LIN {X -91.168,Y -9.449,Z -75.108,A -90.000,B 90.000,C 0.000} C_DIS
LIN {X -91.268,Y -9.455,Z -75.087,A -90.000,B 90.000,C 0.000} C_DIS
LIN {X -91.699,Y -9.484,Z -75.022,A -90.000,B 90.000,C 0.000} C_DIS
LIN {X -91.909,Y -9.497,Z -74.992,A -90.000,B 90.000,C 0.000} C_DIS
LIN {X -92.204,Y -9.516,Z -74.968,A -90.000,B 90.000,C 0.000} C_DIS
LIN {X -92.548,Y -9.529,Z -74.936,A -90.000,B 90.000,C 0.000} C_DIS
LIN {X -93.104,Y -9.554,Z -74.909,A -90.000,B 90.000,C 0.000} C_DIS
LIN {X -93.295,Y -9.561,Z -74.896,A -90.000,B 90.000,C 0.000} C_DIS
LIN {X -93.565,Y -9.563,Z -74.882,A -90.000,B 90.000,C 0.000} C_DIS
LIN {X -93.812,Y -9.568,Z -74.866,A -90.000,B 90.000,C 0.000} C_DIS
LIN {X -94.175,Y -9.581,Z -74.843,A -90.000,B 90.000,C 0.000} C_DIS
LIN {X -94.333,Y -9.590,Z -74.840,A -90.000,B 90.000,C 0.000} C_DIS
LIN {X -94.789,Y -9.599,Z -74.813,A -90.000,B 90.000,C 0.000} C_DIS
LIN {X -95.233,Y -9.601,Z -74.772,A -90.000,B 90.000,C 0.000} C_DIS
LIN {X -95.684,Y -9.621,Z -74.743,A -90.000,B 90.000,C 0.000} C_DIS
LIN {X -95.934,Y -9.627,Z -74.715,A -90.000,B 90.000,C 0.000} C_DIS
LIN {X -95.995,Y -9.627,Z -74.706,A -90.000,B 90.000,C 0.000} C_DIS
LIN {X -96.123,Y -9.624,Z -74.688,A -90.000,B 90.000,C 0.000} C_DIS
LIN {X -96.497,Y -9.616,Z -74.630,A -90.000,B 90.000,C 0.000} C_DIS
LIN {X -96.581,Y -9.616,Z -74.619,A -90.000,B 90.000,C 0.000} C_DIS
LIN {X -96.934,Y -9.624,Z -74.567,A -90.000,B 90.000,C 0.000} C_DIS
LIN {X -97.349,Y -9.643,Z -74.499,A -90.000,B 90.000,C 0.000} C_DIS
LIN {X -97.387,Y -9.643,Z -74.491,A -90.000,B 90.000,C 0.000} C_DIS
LIN {X -97.586,Y -9.638,Z -74.449,A -90.000,B 90.000,C 0.000} C_DIS
LIN {X -97.776,Y -9.630,Z -74.406,A -90.000,B 90.000,C 0.000} C_DIS
LIN {X -97.980,Y -9.623,Z -74.352,A -90.000,B 90.000,C 0.000} C_DIS
LIN {X -98.394,Y -9.618,Z -74.242,A -90.000,B 90.000,C 0.000} C_DIS
LIN {X -98.720,Y -9.626,Z -74.148,A -90.000,B 90.000,C 0.000} C_DIS
LIN {X -99.033,Y -9.638,Z -74.054,A -90.000,B 90.000,C 0.000} C_DIS
LIN {X -99.091,Y -9.639,Z -74.038,A -90.000,B 90.000,C 0.000} C_DIS
LIN {X -99.335,Y -9.635,Z -73.957,A -90.000,B 90.000,C 0.000} C_DIS
LIN {X -99.558,Y -9.626,Z -73.875,A -90.000,B 90.000,C 0.000} C_DIS
LIN {X -99.757,Y -9.620,Z -73.799,A -90.000,B 90.000,C 0.000} C_DIS
LIN {X -100.008,Y -9.607,Z -73.687,A -90.000,B 90.000,C 0.000} C_DIS
LIN {X -100.150,Y -9.603,Z -73.626,A -90.000,B 90.000,C 0.000} C_DIS
LIN {X -100.449,Y -9.604,Z -73.493,A -90.000,B 90.000,C 0.000} C_DIS
LIN {X -100.910,Y -9.619,Z -73.278,A -90.000,B 90.000,C 0.000} C_DIS
LIN {X -101.101,Y -9.624,Z -73.186,A -90.000,B 90.000,C 0.000} C_DIS
LIN {X -101.527,Y -9.617,Z -72.967,A -90.000,B 90.000,C 0.000} C_DIS
LIN {X -101.902,Y -9.589,Z -72.732,A -90.000,B 90.000,C 0.000} C_DIS
LIN {X -101.991,Y -9.585,Z -72.673,A -90.000,B 90.000,C 0.000} C_DIS
LIN {X -102.294,Y -9.577,Z -72.481,A -90.000,B 90.000,C 0.000} C_DIS
LIN {X -102.915,Y -9.585,Z -72.073,A -90.000,B 90.000,C 0.000} C_DIS
LIN {X -103.087,Y -9.586,Z -71.956,A -90.000,B 90.000,C 0.000} C_DIS
LIN {X -103.329,Y -9.590,Z -71.789,A -90.000,B 90.000,C 0.000} C_DIS
LIN {X -104.055,Y -9.563,Z -71.187,A -90.000,B 90.000,C 0.000} C_DIS
LIN {X -104.727,Y -9.571,Z -70.630,A -90.000,B 90.000,C 0.000} C_DIS
LIN {X -105.073,Y -9.578,Z -70.329,A -90.000,B 90.000,C 0.000} C_DIS
LIN {X -105.804,Y -9.557,Z -69.596,A -90.000,B 90.000,C 0.000} C_DIS
LIN {X -106.031,Y -9.558,Z -69.362,A -90.000,B 90.000,C 0.000} C_DIS
LIN {X -106.363,Y -9.567,Z -69.030,A -90.000,B 90.000,C 0.000} C_DIS
LIN {X -106.675,Y -9.569,Z -68.696,A -90.000,B 90.000,C 0.000} C_DIS
LIN {X -107.151,Y -9.555,Z -68.140,A -90.000,B 90.000,C 0.000} C_DIS
LIN {X -107.437,Y -9.551,Z -67.804,A -90.000,B 90.000,C 0.000} C_DIS
LIN {X -107.704,Y -9.554,Z -67.487,A -90.000,B 90.000,C 0.000} C_DIS
LIN {X -107.793,Y -9.554,Z -67.378,A -90.000,B 90.000,C 0.000} C_DIS
LIN {X -108.035,Y -9.548,Z -67.063,A -90.000,B 90.000,C 0.000} C_DIS
LIN {X -108.277,Y -9.542,Z -66.740,A -90.000,B 90.000,C 0.000} C_DIS
LIN {X -108.656,Y -9.536,Z -66.235,A -90.000,B 90.000,C 0.000} C_DIS
LIN {X -109.055,Y -9.536,Z -65.697,A -90.000,B 90.000,C 0.000} C_DIS
LIN {X -109.521,Y -9.515,Z -64.985,A -90.000,B 90.000,C 0.000} C_DIS
LIN {X -109.784,Y -9.507,Z -64.583,A -90.000,B 90.000,C 0.000} C_DIS
LIN {X -109.990,Y -9.509,Z -64.262,A -90.000,B 90.000,C 0.000} C_DIS
LIN {X -110.250,Y -9.507,Z -63.841,A -90.000,B 90.000,C 0.000} C_DIS
LIN {X -110.475,Y -9.498,Z -63.445,A -90.000,B 90.000,C 0.000} C_DIS
LIN {X -110.954,Y -9.484,Z -62.593,A -90.000,B 90.000,C 0.000} C_DIS
LIN {X -111.235,Y -9.477,Z -62.028,A -90.000,B 90.000,C 0.000} C_DIS
LIN {X -111.470,Y -9.467,Z -61.530,A -90.000,B 90.000,C 0.000} C_DIS
LIN {X -111.674,Y -9.468,Z -61.087,A -90.000,B 90.000,C 0.000} C_DIS
LIN {X -111.779,Y -9.472,Z -60.856,A -90.000,B 90.000,C 0.000} C_DIS
LIN {X -111.969,Y -9.471,Z -60.371,A -90.000,B 90.000,C 0.000} C_DIS
LIN {X -112.195,Y -9.468,Z -59.781,A -90.000,B 90.000,C 0.000} C_DIS
LIN {X -112.476,Y -9.471,Z -59.008,A -90.000,B 90.000,C 0.000} C_DIS
LIN {X -112.532,Y -9.474,Z -58.843,A -90.000,B 90.000,C 0.000} C_DIS
LIN {X -112.797,Y -9.477,Z -57.968,A -90.000,B 90.000,C 0.000} C_DIS
LIN {X -112.866,Y -9.485,Z -57.732,A -90.000,B 90.000,C 0.000} C_DIS
LIN {X -112.980,Y -9.499,Z -57.320,A -90.000,B 90.000,C 0.000} C_DIS
LIN {X -113.114,Y -9.515,Z -56.783,A -90.000,B 90.000,C 0.000} C_DIS
LIN {X -113.186,Y -9.521,Z -56.488,A -90.000,B 90.000,C 0.000} C_DIS
LIN {X -113.300,Y -9.536,Z -56.059,A -90.000,B 90.000,C 0.000} C_DIS
LIN {X -113.345,Y -9.541,Z -55.892,A -90.000,B 90.000,C 0.000} C_DIS
LIN {X -113.481,Y -9.549,Z -55.371,A -90.000,B 90.000,C 0.000} C_DIS
LIN {X -113.611,Y -9.568,Z -54.950,A -90.000,B 90.000,C 0.000} C_DIS
LIN {X -113.730,Y -9.575,Z -54.580,A -90.000,B 90.000,C 0.000} C_DIS
LIN {X -113.845,Y -9.584,Z -54.240,A -90.000,B 90.000,C 0.000} C_DIS
LIN {X -113.948,Y -9.588,Z -53.949,A -90.000,B 90.000,C 0.000} C_DIS
LIN {X -114.127,Y -9.591,Z -53.418,A -90.000,B 90.000,C 0.000} C_DIS
LIN {X -114.176,Y -9.591,Z -53.268,A -90.000,B 90.000,C 0.000} C_DIS
LIN {X -114.354,Y -9.592,Z -52.715,A -90.000,B 90.000,C 0.000} C_DIS
LIN {X -114.494,Y -9.589,Z -52.161,A -90.000,B 90.000,C 0.000} C_DIS
LIN {X -114.530,Y -9.591,Z -52.010,A -90.000,B 90.000,C 0.000} C_DIS
LIN {X -114.581,Y -9.592,Z -51.768,A -90.000,B 90.000,C 0.000} C_DIS
LIN {X -114.638,Y -9.569,Z -51.559,A -90.000,B 90.000,C 0.000} C_DIS
LIN {X -114.665,Y -9.552,Z -51.423,A -90.000,B 90.000,C 0.000} C_DIS
LIN {X -114.732,Y -9.507,Z -51.064,A -90.000,B 90.000,C 0.000} C_DIS
LIN {X -114.755,Y -9.494,Z -50.930,A -90.000,B 90.000,C 0.000} C_DIS
LIN {X -114.825,Y -9.450,Z -50.470,A -90.000,B 90.000,C 0.000} C_DIS
LIN {X -114.863,Y -9.414,Z -50.095,A -90.000,B 90.000,C 0.000} C_DIS
LIN {X -114.873,Y -9.404,Z -49.977,A -90.000,B 90.000,C 0.000} C_DIS
LIN {X -115.001,Y -9.414,Z -49.692,A -90.000,B 90.000,C 0.000} C_DIS
LIN {X -115.085,Y -9.419,Z -49.499,A -90.000,B 90.000,C 0.000} C_DIS
LIN {X -115.200,Y -9.434,Z -49.219,A -90.000,B 90.000,C 0.000} C_DIS
LIN {X -115.364,Y -9.456,Z -48.784,A -90.000,B 90.000,C 0.000} C_DIS
LIN {X -115.419,Y -9.463,Z -48.623,A -90.000,B 90.000,C 0.000} C_DIS
LIN {X -115.494,Y -9.476,Z -48.397,A -90.000,B 90.000,C 0.000} C_DIS
LIN {X -115.570,Y -9.486,Z -48.140,A -90.000,B 90.000,C 0.000} C_DIS
LIN {X -115.656,Y -9.511,Z -47.832,A -90.000,B 90.000,C 0.000} C_DIS
LIN {X -115.783,Y -9.545,Z -47.228,A -90.000,B 90.000,C 0.000} C_DIS
LIN {X -115.820,Y -9.560,Z -47.041,A -90.000,B 90.000,C 0.000} C_DIS
LIN {X -115.835,Y -9.566,Z -46.935,A -90.000,B 90.000,C 0.000} C_DIS
LIN {X -115.860,Y -9.577,Z -46.716,A -90.000,B 90.000,C 0.000} C_DIS
LIN {X -115.875,Y -9.588,Z -46.570,A -90.000,B 90.000,C 0.000} C_DIS
LIN {X -115.897,Y -9.607,Z -46.245,A -90.000,B 90.000,C 0.000} C_DIS
LIN {X -115.918,Y -9.644,Z -45.793,A -90.000,B 90.000,C 0.000} C_DIS
LIN {X -115.894,Y -9.672,Z -45.327,A -90.000,B 90.000,C 0.000} C_DIS
LIN {X -115.872,Y -9.694,Z -45.037,A -90.000,B 90.000,C 0.000} C_DIS
LIN {X -115.826,Y -9.720,Z -44.669,A -90.000,B 90.000,C 0.000} C_DIS
LIN {X -115.752,Y -9.743,Z -44.251,A -90.000,B 90.000,C 0.000} C_DIS
LIN {X -115.713,Y -9.747,Z -44.091,A -90.000,B 90.000,C 0.000} C_DIS
LIN {X -115.664,Y -9.757,Z -43.912,A -90.000,B 90.000,C 0.000} C_DIS
LIN {X -115.614,Y -9.765,Z -43.739,A -90.000,B 90.000,C 0.000} C_DIS
LIN {X -115.524,Y -9.782,Z -43.444,A -90.000,B 90.000,C 0.000} C_DIS
LIN {X -115.525,Y -9.755,Z -43.363,A -90.000,B 90.000,C 0.000} C_DIS
LIN {X -115.523,Y -9.708,Z -43.212,A -90.000,B 90.000,C 0.000} C_DIS
LIN {X -115.512,Y -9.657,Z -43.054,A -90.000,B 90.000,C 0.000} C_DIS
LIN {X -115.504,Y -9.620,Z -42.928,A -90.000,B 90.000,C 0.000} C_DIS
LIN {X -115.490,Y -9.576,Z -42.771,A -90.000,B 90.000,C 0.000} C_DIS
LIN {X -115.474,Y -9.541,Z -42.647,A -90.000,B 90.000,C 0.000} C_DIS
LIN {X -115.434,Y -9.476,Z -42.387,A -90.000,B 90.000,C 0.000} C_DIS
LIN {X -115.413,Y -9.451,Z -42.272,A -90.000,B 90.000,C 0.000} C_DIS
LIN {X -115.362,Y -9.404,Z -42.049,A -90.000,B 90.000,C 0.000} C_DIS
LIN {X -115.335,Y -9.385,Z -41.942,A -90.000,B 90.000,C 0.000} C_DIS
LIN {X -115.562,Y -9.395,Z -41.403,A -90.000,B 90.000,C 0.000} C_DIS
LIN {X -115.834,Y -9.409,Z -40.701,A -90.000,B 90.000,C 0.000} C_DIS
LIN {X -115.898,Y -9.411,Z -40.527,A -90.000,B 90.000,C 0.000} C_DIS
LIN {X -115.998,Y -9.421,Z -40.242,A -90.000,B 90.000,C 0.000} C_DIS
LIN {X -116.124,Y -9.434,Z -39.859,A -90.000,B 90.000,C 0.000} C_DIS
LIN {X -116.188,Y -9.437,Z -39.625,A -90.000,B 90.000,C 0.000} C_DIS
LIN {X -116.280,Y -9.448,Z -39.279,A -90.000,B 90.000,C 0.000} C_DIS
LIN {X -116.338,Y -9.459,Z -39.055,A -90.000,B 90.000,C 0.000} C_DIS
LIN {X -116.435,Y -9.475,Z -38.570,A -90.000,B 90.000,C 0.000} C_DIS
LIN {X -116.495,Y -9.485,Z -38.207,A -90.000,B 90.000,C 0.000} C_DIS
LIN {X -116.519,Y -9.488,Z -38.006,A -90.000,B 90.000,C 0.000} C_DIS
LIN {X -116.557,Y -9.499,Z -37.661,A -90.000,B 90.000,C 0.000} C_DIS
LIN {X -116.577,Y -9.508,Z -37.467,A -90.000,B 90.000,C 0.000} C_DIS
LIN {X -116.590,Y -9.517,Z -37.185,A -90.000,B 90.000,C 0.000} C_DIS
LIN {X -116.592,Y -9.520,Z -37.070,A -90.000,B 90.000,C 0.000} C_DIS
LIN {X -116.593,Y -9.528,Z -36.748,A -90.000,B 90.000,C 0.000} C_DIS
LIN {X -116.588,Y -9.536,Z -36.577,A -90.000,B 90.000,C 0.000} C_DIS
LIN {X -116.583,Y -9.544,Z -36.410,A -90.000,B 90.000,C 0.000} C_DIS
LIN {X -116.566,Y -9.555,Z -36.116,A -90.000,B 90.000,C 0.000} C_DIS
LIN {X -116.555,Y -9.557,Z -35.992,A -90.000,B 90.000,C 0.000} C_DIS
LIN {X -116.518,Y -9.569,Z -35.688,A -90.000,B 90.000,C 0.000} C_DIS
LIN {X -116.455,Y -9.588,Z -35.269,A -90.000,B 90.000,C 0.000} C_DIS
LIN {X -116.407,Y -9.596,Z -35.023,A -90.000,B 90.000,C 0.000} C_DIS
LIN {X -116.292,Y -9.604,Z -34.552,A -90.000,B 90.000,C 0.000} C_DIS
LIN {X -116.219,Y -9.613,Z -34.281,A -90.000,B 90.000,C 0.000} C_DIS
LIN {X -116.131,Y -9.620,Z -34.013,A -90.000,B 90.000,C 0.000} C_DIS
LIN {X -115.955,Y -9.626,Z -33.530,A -90.000,B 90.000,C 0.000} C_DIS
LIN {X -115.874,Y -9.632,Z -33.322,A -90.000,B 90.000,C 0.000} C_DIS
LIN {X -115.828,Y -9.634,Z -33.217,A -90.000,B 90.000,C 0.000} C_DIS
LIN {X -115.781,Y -9.638,Z -33.111,A -90.000,B 90.000,C 0.000} C_DIS
LIN {X -115.641,Y -9.647,Z -32.806,A -90.000,B 90.000,C 0.000} C_DIS
LIN {X -115.507,Y -9.653,Z -32.547,A -90.000,B 90.000,C 0.000} C_DIS
LIN {X -115.409,Y -9.659,Z -32.366,A -90.000,B 90.000,C 0.000} C_DIS
LIN {X -115.298,Y -9.671,Z -32.168,A -90.000,B 90.000,C 0.000} C_DIS
LIN {X -115.155,Y -9.677,Z -31.942,A -90.000,B 90.000,C 0.000} C_DIS
LIN {X -114.995,Y -9.683,Z -31.708,A -90.000,B 90.000,C 0.000} C_DIS
LIN {X -114.890,Y -9.691,Z -31.560,A -90.000,B 90.000,C 0.000} C_DIS
LIN {X -114.702,Y -9.699,Z -31.322,A -90.000,B 90.000,C 0.000} C_DIS
LIN {X -114.414,Y -9.707,Z -30.991,A -90.000,B 90.000,C 0.000} C_DIS
LIN {X -114.202,Y -9.712,Z -30.773,A -90.000,B 90.000,C 0.000} C_DIS
LIN {X -113.932,Y -9.710,Z -30.509,A -90.000,B 90.000,C 0.000} C_DIS
LIN {X -113.798,Y -9.696,Z -30.361,A -90.000,B 90.000,C 0.000} C_DIS
LIN {X -113.705,Y -9.684,Z -30.257,A -90.000,B 90.000,C 0.000} C_DIS
LIN {X -113.657,Y -9.679,Z -30.199,A -90.000,B 90.000,C 0.000} C_DIS
LIN {X -113.484,Y -9.675,Z -29.956,A -90.000,B 90.000,C 0.000} C_DIS
LIN {X -113.219,Y -9.679,Z -29.558,A -90.000,B 90.000,C 0.000} C_DIS
LIN {X -112.886,Y -9.691,Z -29.072,A -90.000,B 90.000,C 0.000} C_DIS
LIN {X -112.575,Y -9.712,Z -28.647,A -90.000,B 90.000,C 0.000} C_DIS
LIN {X -112.441,Y -9.714,Z -28.475,A -90.000,B 90.000,C 0.000} C_DIS
LIN {X -112.214,Y -9.724,Z -28.195,A -90.000,B 90.000,C 0.000} C_DIS
LIN {X -111.965,Y -9.730,Z -27.908,A -90.000,B 90.000,C 0.000} C_DIS
LIN {X -111.767,Y -9.733,Z -27.682,A -90.000,B 90.000,C 0.000} C_DIS
LIN {X -111.552,Y -9.744,Z -27.448,A -90.000,B 90.000,C 0.000} C_DIS
LIN {X -111.335,Y -9.745,Z -27.227,A -90.000,B 90.000,C 0.000} C_DIS
LIN {X -111.169,Y -9.752,Z -27.063,A -90.000,B 90.000,C 0.000} C_DIS
LIN {X -110.868,Y -9.756,Z -26.783,A -90.000,B 90.000,C 0.000} C_DIS
LIN {X -110.555,Y -9.759,Z -26.498,A -90.000,B 90.000,C 0.000} C_DIS
LIN {X -110.409,Y -9.764,Z -26.368,A -90.000,B 90.000,C 0.000} C_DIS
LIN {X -110.072,Y -9.763,Z -26.089,A -90.000,B 90.000,C 0.000} C_DIS
LIN {X -109.993,Y -9.765,Z -26.026,A -90.000,B 90.000,C 0.000} C_DIS
LIN {X -109.797,Y -9.772,Z -25.877,A -90.000,B 90.000,C 0.000} C_DIS
LIN {X -109.647,Y -9.773,Z -25.770,A -90.000,B 90.000,C 0.000} C_DIS
LIN {X -109.156,Y -9.772,Z -25.430,A -90.000,B 90.000,C 0.000} C_DIS
LIN {X -109.060,Y -9.773,Z -25.365,A -90.000,B 90.000,C 0.000} C_DIS
LIN {X -108.938,Y -9.779,Z -25.289,A -90.000,B 90.000,C 0.000} C_DIS
LIN {X -108.645,Y -9.778,Z -25.128,A -90.000,B 90.000,C 0.000} C_DIS
LIN {X -107.965,Y -9.778,Z -24.760,A -90.000,B 90.000,C 0.000} C_DIS
LIN {X -107.894,Y -9.777,Z -24.729,A -90.000,B 90.000,C 0.000} C_DIS
LIN {X -107.430,Y -9.777,Z -24.533,A -90.000,B 90.000,C 0.000} C_DIS
LIN {X -107.064,Y -9.775,Z -24.380,A -90.000,B 90.000,C 0.000} C_DIS
LIN {X -106.859,Y -9.774,Z -24.300,A -90.000,B 90.000,C 0.000} C_DIS
LIN {X -106.675,Y -9.768,Z -24.235,A -90.000,B 90.000,C 0.000} C_DIS
LIN {X -105.951,Y -9.767,Z -23.999,A -90.000,B 90.000,C 0.000} C_DIS
LIN {X -105.833,Y -9.766,Z -23.963,A -90.000,B 90.000,C 0.000} C_DIS
LIN {X -105.591,Y -9.759,Z -23.893,A -90.000,B 90.000,C 0.000} C_DIS
LIN {X -104.540,Y -9.751,Z -23.612,A -90.000,B 90.000,C 0.000} C_DIS
LIN {X -104.007,Y -9.738,Z -23.487,A -90.000,B 90.000,C 0.000} C_DIS
LIN {X -103.457,Y -9.732,Z -23.351,A -90.000,B 90.000,C 0.000} C_DIS
LIN {X -102.983,Y -9.716,Z -23.250,A -90.000,B 90.000,C 0.000} C_DIS
LIN {X -102.872,Y -9.662,Z -23.190,A -90.000,B 90.000,C 0.000} C_DIS
LIN {X -102.791,Y -9.626,Z -23.147,A -90.000,B 90.000,C 0.000} C_DIS
LIN {X -102.651,Y -9.570,Z -23.076,A -90.000,B 90.000,C 0.000} C_DIS
LIN {X -102.484,Y -9.509,Z -22.997,A -90.000,B 90.000,C 0.000} C_DIS
LIN {X -102.347,Y -9.465,Z -22.940,A -90.000,B 90.000,C 0.000} C_DIS
LIN {X -102.173,Y -9.419,Z -22.874,A -90.000,B 90.000,C 0.000} C_DIS
LIN {X -102.051,Y -9.391,Z -22.833,A -90.000,B 90.000,C 0.000} C_DIS
LIN {X -101.981,Y -9.396,Z -22.678,A -90.000,B 90.000,C 0.000} C_DIS
LIN {X -101.915,Y -9.397,Z -22.554,A -90.000,B 90.000,C 0.000} C_DIS
LIN {X -101.706,Y -9.412,Z -22.179,A -90.000,B 90.000,C 0.000} C_DIS
LIN {X -101.652,Y -9.413,Z -22.097,A -90.000,B 90.000,C 0.000} C_DIS
LIN {X -101.407,Y -9.417,Z -21.742,A -90.000,B 90.000,C 0.000} C_DIS
LIN {X -101.220,Y -9.429,Z -21.478,A -90.000,B 90.000,C 0.000} C_DIS
LIN {X -101.124,Y -9.431,Z -21.364,A -90.000,B 90.000,C 0.000} C_DIS
LIN {X -100.916,Y -9.439,Z -21.124,A -90.000,B 90.000,C 0.000} C_DIS
LIN {X -100.729,Y -9.441,Z -20.929,A -90.000,B 90.000,C 0.000} C_DIS
LIN {X -100.489,Y -9.453,Z -20.691,A -90.000,B 90.000,C 0.000} C_DIS
LIN {X -100.427,Y -9.456,Z -20.633,A -90.000,B 90.000,C 0.000} C_DIS
LIN {X -100.372,Y -9.456,Z -20.587,A -90.000,B 90.000,C 0.000} C_DIS
LIN {X -100.028,Y -9.469,Z -20.310,A -90.000,B 90.000,C 0.000} C_DIS
LIN {X -99.660,Y -9.482,Z -20.039,A -90.000,B 90.000,C 0.000} C_DIS
LIN {X -99.572,Y -9.484,Z -19.982,A -90.000,B 90.000,C 0.000} C_DIS
LIN {X -99.263,Y -9.501,Z -19.787,A -90.000,B 90.000,C 0.000} C_DIS
LIN {X -99.057,Y -9.514,Z -19.661,A -90.000,B 90.000,C 0.000} C_DIS
LIN {X -98.687,Y -9.550,Z -19.438,A -90.000,B 90.000,C 0.000} C_DIS
LIN {X -98.564,Y -9.558,Z -19.362,A -90.000,B 90.000,C 0.000} C_DIS
LIN {X -98.513,Y -9.563,Z -19.327,A -90.000,B 90.000,C 0.000} C_DIS
LIN {X -98.444,Y -9.564,Z -19.279,A -90.000,B 90.000,C 0.000} C_DIS
LIN {X -98.167,Y -9.553,Z -19.075,A -90.000,B 90.000,C 0.000} C_DIS
LIN {X -97.827,Y -9.534,Z -18.818,A -90.000,B 90.000,C 0.000} C_DIS
LIN {X -97.309,Y -9.513,Z -18.416,A -90.000,B 90.000,C 0.000} C_DIS
LIN {X -96.939,Y -9.494,Z -18.137,A -90.000,B 90.000,C 0.000} C_DIS
LIN {X -96.775,Y -9.486,Z -18.015,A -90.000,B 90.000,C 0.000} C_DIS
LIN {X -96.559,Y -9.477,Z -17.860,A -90.000,B 90.000,C 0.000} C_DIS
LIN {X -96.169,Y -9.461,Z -17.597,A -90.000,B 90.000,C 0.000} C_DIS
LIN {X -96.082,Y -9.456,Z -17.542,A -90.000,B 90.000,C 0.000} C_DIS
LIN {X -95.833,Y -9.448,Z -17.385,A -90.000,B 90.000,C 0.000} C_DIS
LIN {X -95.570,Y -9.443,Z -17.225,A -90.000,B 90.000,C 0.000} C_DIS
LIN {X -95.432,Y -9.438,Z -17.152,A -90.000,B 90.000,C 0.000} C_DIS
LIN {X -95.237,Y -9.434,Z -17.050,A -90.000,B 90.000,C 0.000} C_DIS
LIN {X -94.597,Y -9.418,Z -16.733,A -90.000,B 90.000,C 0.000} C_DIS
LIN {X -94.412,Y -9.417,Z -16.644,A -90.000,B 90.000,C 0.000} C_DIS
LIN {X -94.337,Y -9.418,Z -16.611,A -90.000,B 90.000,C 0.000} C_DIS
LIN {X -93.696,Y -9.405,Z -16.376,A -90.000,B 90.000,C 0.000} C_DIS
LIN {X -93.310,Y -9.397,Z -16.248,A -90.000,B 90.000,C 0.000} C_DIS
LIN {X -93.123,Y -9.398,Z -16.184,A -90.000,B 90.000,C 0.000} C_DIS
LIN {X -92.656,Y -9.392,Z -16.067,A -90.000,B 90.000,C 0.000} C_DIS
LIN {X -91.926,Y -9.379,Z -15.911,A -90.000,B 90.000,C 0.000} C_DIS
LIN {X -91.743,Y -9.379,Z -15.873,A -90.000,B 90.000,C 0.000} C_DIS
LIN {X -91.620,Y -9.377,Z -15.856,A -90.000,B 90.000,C 0.000} C_DIS
LIN {X -91.266,Y -9.374,Z -15.806,A -90.000,B 90.000,C 0.000} C_DIS
LIN {X -90.401,Y -9.364,Z -15.706,A -90.000,B 90.000,C 0.000} C_DIS
LIN {X -90.201,Y -9.365,Z -15.684,A -90.000,B 90.000,C 0.000} C_DIS
LIN {X -89.078,Y -9.360,Z -15.638,A -90.000,B 90.000,C 0.000} C_DIS
LIN {X -88.674,Y -9.357,Z -15.629,A -90.000,B 90.000,C 0.000} C_DIS
LIN {X -88.466,Y -9.360,Z -15.627,A -90.000,B 90.000,C 0.000} C_DIS
LIN {X -87.996,Y -9.370,Z -15.609,A -90.000,B 90.000,C 0.000} C_DIS
LIN {X -87.769,Y -9.388,Z -15.554,A -90.000,B 90.000,C 0.000} C_DIS
LIN {X -87.406,Y -9.434,Z -15.431,A -90.000,B 90.000,C 0.000} C_DIS
LIN {X -87.259,Y -9.455,Z -15.384,A -90.000,B 90.000,C 0.000} C_DIS
LIN {X -87.086,Y -9.435,Z -15.291,A -90.000,B 90.000,C 0.000} C_DIS
LIN {X -86.910,Y -9.416,Z -15.206,A -90.000,B 90.000,C 0.000} C_DIS
LIN {X -86.634,Y -9.396,Z -15.047,A -90.000,B 90.000,C 0.000} C_DIS
LIN {X -86.363,Y -9.385,Z -14.877,A -90.000,B 90.000,C 0.000} C_DIS
LIN {X -86.283,Y -9.382,Z -14.831,A -90.000,B 90.000,C 0.000} C_DIS
LIN {X -85.944,Y -9.369,Z -14.637,A -90.000,B 90.000,C 0.000} C_DIS
LIN {X -85.650,Y -9.362,Z -14.473,A -90.000,B 90.000,C 0.000} C_DIS
LIN {X -85.531,Y -9.359,Z -14.412,A -90.000,B 90.000,C 0.000} C_DIS
LIN {X -85.166,Y -9.354,Z -14.243,A -90.000,B 90.000,C 0.000} C_DIS
LIN {X -85.013,Y -9.352,Z -14.175,A -90.000,B 90.000,C 0.000} C_DIS
LIN {X -84.538,Y -9.350,Z -13.956,A -90.000,B 90.000,C 0.000} C_DIS
LIN {X -84.494,Y -9.349,Z -13.939,A -90.000,B 90.000,C 0.000} C_DIS
LIN {X -84.021,Y -9.344,Z -13.777,A -90.000,B 90.000,C 0.000} C_DIS
LIN {X -83.767,Y -9.341,Z -13.708,A -90.000,B 90.000,C 0.000} C_DIS
LIN {X -83.266,Y -9.348,Z -13.537,A -90.000,B 90.000,C 0.000} C_DIS
LIN {X -82.789,Y -9.343,Z -13.426,A -90.000,B 90.000,C 0.000} C_DIS
LIN {X -82.461,Y -9.340,Z -13.367,A -90.000,B 90.000,C 0.000} C_DIS
LIN {X -82.347,Y -9.342,Z -13.339,A -90.000,B 90.000,C 0.000} C_DIS
LIN {X -81.876,Y -9.348,Z -13.231,A -90.000,B 90.000,C 0.000} C_DIS
LIN {X -81.752,Y -9.347,Z -13.212,A -90.000,B 90.000,C 0.000} C_DIS
LIN {X -81.565,Y -9.344,Z -13.188,A -90.000,B 90.000,C 0.000} C_DIS
LIN {X -81.150,Y -9.342,Z -13.137,A -90.000,B 90.000,C 0.000} C_DIS
LIN {X -80.838,Y -9.345,Z -13.089,A -90.000,B 90.000,C 0.000} C_DIS
LIN {X -80.305,Y -9.348,Z -13.023,A -90.000,B 90.000,C 0.000} C_DIS
LIN {X -80.034,Y -9.345,Z -13.005,A -90.000,B 90.000,C 0.000} C_DIS
LIN {X -79.553,Y -9.341,Z -12.994,A -90.000,B 90.000,C 0.000} C_DIS
LIN {X -79.360,Y -9.341,Z -12.989,A -90.000,B 90.000,C 0.000} C_DIS
LIN {X -78.738,Y -9.342,Z -12.974,A -90.000,B 90.000,C 0.000} C_DIS
LIN {X -78.639,Y -9.341,Z -12.980,A -90.000,B 90.000,C 0.000} C_DIS
LIN {X -78.208,Y -9.337,Z -13.002,A -90.000,B 90.000,C 0.000} C_DIS
LIN {X -77.711,Y -9.335,Z -13.042,A -90.000,B 90.000,C 0.000} C_DIS
LIN {X -77.209,Y -9.333,Z -13.099,A -90.000,B 90.000,C 0.000} C_DIS
LIN {X -76.730,Y -9.330,Z -13.189,A -90.000,B 90.000,C 0.000} C_DIS
LIN {X -76.215,Y -9.325,Z -13.317,A -90.000,B 90.000,C 0.000} C_DIS
LIN {X -75.542,Y -9.324,Z -13.472,A -90.000,B 90.000,C 0.000} C_DIS
LIN {X -75.075,Y -9.322,Z -13.609,A -90.000,B 90.000,C 0.000} C_DIS
LIN {X -74.485,Y -9.319,Z -13.813,A -90.000,B 90.000,C 0.000} C_DIS
LIN {X -74.204,Y -9.320,Z -13.917,A -90.000,B 90.000,C 0.000} C_DIS
LIN {X -74.078,Y -9.321,Z -13.959,A -90.000,B 90.000,C 0.000} C_DIS
LIN {X -73.706,Y -9.320,Z -14.113,A -90.000,B 90.000,C 0.000} C_DIS
LIN {X -73.440,Y -9.319,Z -14.227,A -90.000,B 90.000,C 0.000} C_DIS
LIN {X -72.817,Y -9.320,Z -14.463,A -90.000,B 90.000,C 0.000} C_DIS
LIN {X -72.241,Y -9.321,Z -14.699,A -90.000,B 90.000,C 0.000} C_DIS
LIN {X -71.159,Y -9.322,Z -15.152,A -90.000,B 90.000,C 0.000} C_DIS
LIN {X -70.148,Y -9.324,Z -15.584,A -90.000,B 90.000,C 0.000} C_DIS
LIN {X -69.794,Y -9.326,Z -15.729,A -90.000,B 90.000,C 0.000} C_DIS
LIN {X -69.695,Y -9.327,Z -15.770,A -90.000,B 90.000,C 0.000} C_DIS
LIN {X -68.555,Y -9.332,Z -16.265,A -90.000,B 90.000,C 0.000} C_DIS
LIN {X -68.227,Y -9.335,Z -16.400,A -90.000,B 90.000,C 0.000} C_DIS
LIN {X -67.078,Y -9.342,Z -16.902,A -90.000,B 90.000,C 0.000} C_DIS
LIN {X -66.779,Y -9.345,Z -17.026,A -90.000,B 90.000,C 0.000} C_DIS
LIN {X -66.334,Y -9.348,Z -17.219,A -90.000,B 90.000,C 0.000} C_DIS
LIN {X -66.228,Y -9.355,Z -17.231,A -90.000,B 90.000,C 0.000} C_DIS
LIN {X -65.840,Y -9.380,Z -17.303,A -90.000,B 90.000,C 0.000} C_DIS
LIN {X -65.586,Y -9.399,Z -17.350,A -90.000,B 90.000,C 0.000} C_DIS
LIN {X -64.905,Y -9.455,Z -17.485,A -90.000,B 90.000,C 0.000} C_DIS
LIN {X -64.585,Y -9.481,Z -17.559,A -90.000,B 90.000,C 0.000} C_DIS
LIN {X -64.137,Y -9.519,Z -17.672,A -90.000,B 90.000,C 0.000} C_DIS
LIN {X -64.046,Y -9.527,Z -17.697,A -90.000,B 90.000,C 0.000} C_DIS
LIN {X -63.342,Y -9.588,Z -17.879,A -90.000,B 90.000,C 0.000} C_DIS
LIN {X -62.974,Y -9.620,Z -17.978,A -90.000,B 90.000,C 0.000} C_DIS
LIN {X -62.811,Y -9.635,Z -18.025,A -90.000,B 90.000,C 0.000} C_DIS
LIN {X -62.330,Y -9.677,Z -18.156,A -90.000,B 90.000,C 0.000} C_DIS
LIN {X -61.465,Y -9.767,Z -18.380,A -90.000,B 90.000,C 0.000} C_DIS
LIN {X -61.175,Y -9.806,Z -18.445,A -90.000,B 90.000,C 0.000} C_DIS
LIN {X -60.456,Y -9.908,Z -18.613,A -90.000,B 90.000,C 0.000} C_DIS
LIN {X -60.042,Y -9.974,Z -18.704,A -90.000,B 90.000,C 0.000} C_DIS
LIN {X -59.718,Y -10.030,Z -18.781,A -90.000,B 90.000,C 0.000} C_DIS
LIN {X -59.320,Y -10.090,Z -18.863,A -90.000,B 90.000,C 0.000} C_DIS
LIN {X -58.810,Y -10.173,Z -18.980,A -90.000,B 90.000,C 0.000} C_DIS
LIN {X -58.277,Y -10.249,Z -19.087,A -90.000,B 90.000,C 0.000} C_DIS
LIN {X -57.905,Y -10.296,Z -19.168,A -90.000,B 90.000,C 0.000} C_DIS
LIN {X -57.193,Y -10.363,Z -19.289,A -90.000,B 90.000,C 0.000} C_DIS
LIN {X -56.927,Y -10.383,Z -19.336,A -90.000,B 90.000,C 0.000} C_DIS
LIN {X -56.708,Y -10.378,Z -19.345,A -90.000,B 90.000,C 0.000} C_DIS
LIN {X -56.307,Y -10.365,Z -19.364,A -90.000,B 90.000,C 0.000} C_DIS
LIN {X -56.081,Y -10.358,Z -19.375,A -90.000,B 90.000,C 0.000} C_DIS
LIN {X -55.759,Y -10.345,Z -19.387,A -90.000,B 90.000,C 0.000} C_DIS
LIN {X -55.661,Y -10.343,Z -19.392,A -90.000,B 90.000,C 0.000} C_DIS
LIN {X -55.218,Y -10.340,Z -19.429,A -90.000,B 90.000,C 0.000} C_DIS
LIN {X -54.399,Y -10.319,Z -19.507,A -90.000,B 90.000,C 0.000} C_DIS
LIN {X -53.422,Y -10.292,Z -19.607,A -90.000,B 90.000,C 0.000} C_DIS
LIN {X -53.081,Y -10.280,Z -19.652,A -90.000,B 90.000,C 0.000} C_DIS
LIN {X -51.231,Y -10.230,Z -19.890,A -90.000,B 90.000,C 0.000} C_DIS
LIN {X -49.816,Y -10.185,Z -20.090,A -90.000,B 90.000,C 0.000} C_DIS
LIN {X -48.591,Y -10.155,Z -20.272,A -90.000,B 90.000,C 0.000} C_DIS
LIN {X -47.049,Y -10.125,Z -20.505,A -90.000,B 90.000,C 0.000} C_DIS
LIN {X -45.652,Y -10.083,Z -20.700,A -90.000,B 90.000,C 0.000} C_DIS
LIN {X -45.519,Y -10.076,Z -20.720,A -90.000,B 90.000,C 0.000} C_DIS
LIN {X -43.641,Y -10.019,Z -21.048,A -90.000,B 90.000,C 0.000} C_DIS
LIN {X -43.412,Y -10.010,Z -21.089,A -90.000,B 90.000,C 0.000} C_DIS
LIN {X -42.448,Y -9.983,Z -21.284,A -90.000,B 90.000,C 0.000} C_DIS
LIN {X -41.810,Y -9.964,Z -21.396,A -90.000,B 90.000,C 0.000} C_DIS
LIN {X -40.603,Y -9.929,Z -21.625,A -90.000,B 90.000,C 0.000} C_DIS
LIN {X -40.430,Y -9.921,Z -21.655,A -90.000,B 90.000,C 0.000} C_DIS
LIN {X -39.323,Y -9.889,Z -21.832,A -90.000,B 90.000,C 0.000} C_DIS
LIN {X -38.147,Y -9.877,Z -22.040,A -90.000,B 90.000,C 0.000} C_DIS
LIN {X -36.836,Y -9.849,Z -22.289,A -90.000,B 90.000,C 0.000} C_DIS
LIN {X -35.421,Y -9.843,Z -22.578,A -90.000,B 90.000,C 0.000} C_DIS
LIN {X -35.170,Y -9.840,Z -22.632,A -90.000,B 90.000,C 0.000} C_DIS
LIN {X -34.760,Y -9.830,Z -22.717,A -90.000,B 90.000,C 0.000} C_DIS
LIN {X -34.476,Y -9.826,Z -22.773,A -90.000,B 90.000,C 0.000} C_DIS
LIN {X -33.387,Y -9.805,Z -22.998,A -90.000,B 90.000,C 0.000} C_DIS
LIN {X -31.836,Y -9.778,Z -23.322,A -90.000,B 90.000,C 0.000} C_DIS
LIN {X -30.713,Y -9.763,Z -23.550,A -90.000,B 90.000,C 0.000} C_DIS
LIN {X -29.647,Y -9.745,Z -23.772,A -90.000,B 90.000,C 0.000} C_DIS
LIN {X -27.374,Y -9.720,Z -24.252,A -90.000,B 90.000,C 0.000} C_DIS
LIN {X -26.770,Y -9.713,Z -24.381,A -90.000,B 90.000,C 0.000} C_DIS
LIN {X -22.896,Y -9.701,Z -25.233,A -90.000,B 90.000,C 0.000} C_DIS
LIN {X -20.698,Y -9.690,Z -25.738,A -90.000,B 90.000,C 0.000} C_DIS
LIN {X -18.278,Y -9.682,Z -26.292,A -90.000,B 90.000,C 0.000} C_DIS
LIN {X -17.330,Y -9.678,Z -26.506,A -90.000,B 90.000,C 0.000} C_DIS
LIN {X -15.885,Y -9.675,Z -26.837,A -90.000,B 90.000,C 0.000} C_DIS
LIN {X -12.820,Y -9.659,Z -27.520,A -90.000,B 90.000,C 0.000} C_DIS
LIN {X -11.931,Y -9.656,Z -27.721,A -90.000,B 90.000,C 0.000} C_DIS
LIN {X -9.515,Y -9.643,Z -28.245,A -90.000,B 90.000,C 0.000} C_DIS
LIN {X -8.971,Y -9.640,Z -28.365,A -90.000,B 90.000,C 0.000} C_DIS
LIN {X -6.728,Y -9.646,Z -28.839,A -90.000,B 90.000,C 0.000} C_DIS
LIN {X -5.891,Y -9.645,Z -29.019,A -90.000,B 90.000,C 0.000} C_DIS
LIN {X -4.975,Y -9.643,Z -29.202,A -90.000,B 90.000,C 0.000} C_DIS
LIN {X -3.552,Y -9.643,Z -29.489,A -90.000,B 90.000,C 0.000} C_DIS
LIN {X -2.855,Y -9.640,Z -29.634,A -90.000,B 90.000,C 0.000} C_DIS
LIN {X -1.549,Y -9.637,Z -29.882,A -90.000,B 90.000,C 0.000} C_DIS
LIN {X -0.835,Y -9.630,Z -30.014,A -90.000,B 90.000,C 0.000} C_DIS
LIN {X -0.170,Y -9.626,Z -30.132,A -90.000,B 90.000,C 0.000} C_DIS
LIN {X 0.860,Y -9.623,Z -30.317,A -90.000,B 90.000,C 0.000} C_DIS
LIN {X 1.585,Y -9.615,Z -30.444,A -90.000,B 90.000,C 0.000} C_DIS
LIN {X 2.719,Y -9.611,Z -30.626,A -90.000,B 90.000,C 0.000} C_DIS
LIN {X 2.859,Y -9.609,Z -30.651,A -90.000,B 90.000,C 0.000} C_DIS
LIN {X 3.240,Y -9.609,Z -30.720,A -90.000,B 90.000,C 0.000} C_DIS
LIN {X 3.941,Y -9.601,Z -30.844,A -90.000,B 90.000,C 0.000} C_DIS
LIN {X 5.105,Y -9.600,Z -31.029,A -90.000,B 90.000,C 0.000} C_DIS
LIN {X 5.458,Y -9.603,Z -31.086,A -90.000,B 90.000,C 0.000} C_DIS
LIN {X 5.600,Y -9.601,Z -31.114,A -90.000,B 90.000,C 0.000} C_DIS
LIN {X 6.205,Y -9.600,Z -31.235,A -90.000,B 90.000,C 0.000} C_DIS
LIN {X 7.941,Y -9.622,Z -31.545,A -90.000,B 90.000,C 0.000} C_DIS
LIN {X 8.237,Y -9.622,Z -31.596,A -90.000,B 90.000,C 0.000} C_DIS
LIN {X 8.641,Y -9.622,Z -31.681,A -90.000,B 90.000,C 0.000} C_DIS
LIN {X 10.572,Y -9.641,Z -32.103,A -90.000,B 90.000,C 0.000} C_DIS
LIN {X 11.267,Y -9.639,Z -32.264,A -90.000,B 90.000,C 0.000} C_DIS
LIN {X 11.987,Y -9.646,Z -32.435,A -90.000,B 90.000,C 0.000} C_DIS
LIN {X 12.666,Y -9.649,Z -32.601,A -90.000,B 90.000,C 0.000} C_DIS
LIN {X 13.445,Y -9.645,Z -32.778,A -90.000,B 90.000,C 0.000} C_DIS
LIN {X 14.264,Y -9.647,Z -32.969,A -90.000,B 90.000,C 0.000} C_DIS
LIN {X 14.518,Y -9.654,Z -33.020,A -90.000,B 90.000,C 0.000} C_DIS
LIN {X 15.683,Y -9.651,Z -33.236,A -90.000,B 90.000,C 0.000} C_DIS
LIN {X 15.945,Y -9.657,Z -33.273,A -90.000,B 90.000,C 0.000} C_DIS
LIN {X 16.523,Y -9.655,Z -33.333,A -90.000,B 90.000,C 0.000} C_DIS
LIN {X 17.296,Y -9.641,Z -33.404,A -90.000,B 90.000,C 0.000} C_DIS
LIN {X 17.590,Y -9.642,Z -33.417,A -90.000,B 90.000,C 0.000} C_DIS
LIN {X 18.416,Y -9.614,Z -33.438,A -90.000,B 90.000,C 0.000} C_DIS
LIN {X 18.547,Y -9.610,Z -33.446,A -90.000,B 90.000,C 0.000} C_DIS
LIN {X 18.729,Y -9.609,Z -33.448,A -90.000,B 90.000,C 0.000} C_DIS
LIN {X 19.569,Y -9.577,Z -33.441,A -90.000,B 90.000,C 0.000} C_DIS
LIN {X 19.804,Y -9.570,Z -33.441,A -90.000,B 90.000,C 0.000} C_DIS
LIN {X 20.946,Y -9.528,Z -33.445,A -90.000,B 90.000,C 0.000} C_DIS
LIN {X 21.432,Y -9.519,Z -33.450,A -90.000,B 90.000,C 0.000} C_DIS
LIN {X 21.614,Y -9.516,Z -33.456,A -90.000,B 90.000,C 0.000} C_DIS
LIN {X 22.698,Y -9.488,Z -33.517,A -90.000,B 90.000,C 0.000} C_DIS
LIN {X 23.071,Y -9.486,Z -33.540,A -90.000,B 90.000,C 0.000} C_DIS
LIN {X 24.102,Y -9.468,Z -33.643,A -90.000,B 90.000,C 0.000} C_DIS
LIN {X 24.296,Y -9.464,Z -33.666,A -90.000,B 90.000,C 0.000} C_DIS
LIN {X 24.544,Y -9.461,Z -33.697,A -90.000,B 90.000,C 0.000} C_DIS
LIN {X 24.933,Y -9.452,Z -33.755,A -90.000,B 90.000,C 0.000} C_DIS
LIN {X 25.584,Y -9.439,Z -33.859,A -90.000,B 90.000,C 0.000} C_DIS
LIN {X 26.136,Y -9.432,Z -33.949,A -90.000,B 90.000,C 0.000} C_DIS
LIN {X 26.539,Y -9.427,Z -34.018,A -90.000,B 90.000,C 0.000} C_DIS
LIN {X 27.360,Y -9.413,Z -34.177,A -90.000,B 90.000,C 0.000} C_DIS
LIN {X 27.758,Y -9.408,Z -34.256,A -90.000,B 90.000,C 0.000} C_DIS
LIN {X 28.112,Y -9.404,Z -34.330,A -90.000,B 90.000,C 0.000} C_DIS
LIN {X 28.830,Y -9.392,Z -34.495,A -90.000,B 90.000,C 0.000} C_DIS
LIN {X 29.830,Y -9.378,Z -34.717,A -90.000,B 90.000,C 0.000} C_DIS
LIN {X 31.584,Y -9.352,Z -35.156,A -90.000,B 90.000,C 0.000} C_DIS
LIN {X 32.299,Y -9.343,Z -35.348,A -90.000,B 90.000,C 0.000} C_DIS
LIN {X 33.525,Y -9.331,Z -35.681,A -90.000,B 90.000,C 0.000} C_DIS
LIN {X 34.181,Y -9.324,Z -35.875,A -90.000,B 90.000,C 0.000} C_DIS
LIN {X 35.875,Y -9.314,Z -36.394,A -90.000,B 90.000,C 0.000} C_DIS
LIN {X 36.548,Y -9.312,Z -36.610,A -90.000,B 90.000,C 0.000} C_DIS
LIN {X 38.957,Y -9.308,Z -37.388,A -90.000,B 90.000,C 0.000} C_DIS
LIN {X 39.464,Y -9.308,Z -37.560,A -90.000,B 90.000,C 0.000} C_DIS
LIN {X 39.464,Y -60.000,Z -37.560,A -90.000,B 90.000,C 0.000} C_DIS
LIN {X 49.651,Y -60.000,Z -41.198,A -90.000,B 90.000,C 0.000} C_DIS
LIN {X 49.651,Y -9.308,Z -41.198,A -90.000,B 90.000,C 0.000} C_DIS
LIN {X 49.716,Y -9.308,Z -41.231,A -90.000,B 90.000,C 0.000} C_DIS
LIN {X 49.716,Y -60.000,Z -41.231,A -90.000,B 90.000,C 0.000} C_DIS
LIN {X 58.412,Y -60.000,Z -46.839,A -90.000,B 90.000,C 0.000} C_DIS
LIN {X 58.412,Y -9.308,Z -46.839,A -90.000,B 90.000,C 0.000} C_DIS
LIN {X 58.604,Y -9.309,Z -46.948,A -90.000,B 90.000,C 0.000} C_DIS
LIN {X 59.663,Y -9.337,Z -47.460,A -90.000,B 90.000,C 0.000} C_DIS
LIN {X 60.145,Y -9.343,Z -47.692,A -90.000,B 90.000,C 0.000} C_DIS
LIN {X 60.503,Y -9.345,Z -47.880,A -90.000,B 90.000,C 0.000} C_DIS
LIN {X 61.492,Y -9.348,Z -48.418,A -90.000,B 90.000,C 0.000} C_DIS
LIN {X 62.933,Y -9.357,Z -49.110,A -90.000,B 90.000,C 0.000} C_DIS
LIN {X 63.624,Y -9.358,Z -49.455,A -90.000,B 90.000,C 0.000} C_DIS
LIN {X 64.812,Y -9.357,Z -50.046,A -90.000,B 90.000,C 0.000} C_DIS
LIN {X 65.266,Y -9.358,Z -50.271,A -90.000,B 90.000,C 0.000} C_DIS
LIN {X 65.873,Y -9.358,Z -50.581,A -90.000,B 90.000,C 0.000} C_DIS
LIN {X 66.591,Y -9.356,Z -50.956,A -90.000,B 90.000,C 0.000} C_DIS
LIN {X 67.150,Y -9.355,Z -51.255,A -90.000,B 90.000,C 0.000} C_DIS
LIN {X 67.828,Y -9.357,Z -51.618,A -90.000,B 90.000,C 0.000} C_DIS
LIN {X 68.013,Y -9.357,Z -51.721,A -90.000,B 90.000,C 0.000} C_DIS
LIN {X 68.612,Y -9.355,Z -52.065,A -90.000,B 90.000,C 0.000} C_DIS
LIN {X 69.520,Y -9.352,Z -52.587,A -90.000,B 90.000,C 0.000} C_DIS
LIN {X 70.507,Y -9.349,Z -53.184,A -90.000,B 90.000,C 0.000} C_DIS
LIN {X 71.379,Y -9.348,Z -53.709,A -90.000,B 90.000,C 0.000} C_DIS
LIN {X 73.487,Y -9.346,Z -55.032,A -90.000,B 90.000,C 0.000} C_DIS
LIN {X 75.401,Y -9.347,Z -56.275,A -90.000,B 90.000,C 0.000} C_DIS
LIN {X 75.810,Y -9.348,Z -56.545,A -90.000,B 90.000,C 0.000} C_DIS
LIN {X 77.661,Y -9.354,Z -57.793,A -90.000,B 90.000,C 0.000} C_DIS
LIN {X 77.914,Y -9.357,Z -57.967,A -90.000,B 90.000,C 0.000} C_DIS
LIN {X 78.796,Y -9.362,Z -58.602,A -90.000,B 90.000,C 0.000} C_DIS
LIN {X 78.945,Y -9.363,Z -58.709,A -90.000,B 90.000,C 0.000} C_DIS
LIN {X 79.461,Y -9.367,Z -59.080,A -90.000,B 90.000,C 0.000} C_DIS
LIN {X 79.825,Y -9.369,Z -59.336,A -90.000,B 90.000,C 0.000} C_DIS
LIN {X 79.826,Y -17.867,Z -59.337,A -90.000,B 90.000,C 0.000} C_DIS
LIN {X 79.831,Y -18.015,Z -59.340,A -90.000,B 90.000,C 0.000} C_DIS
LIN {X 79.878,Y -18.662,Z -59.372,A -90.000,B 90.000,C 0.000} C_DIS
LIN {X 79.968,Y -19.143,Z -59.433,A -90.000,B 90.000,C 0.000} C_DIS
LIN {X 80.053,Y -19.414,Z -59.489,A -90.000,B 90.000,C 0.000} C_DIS
LIN {X 80.133,Y -19.543,Z -59.541,A -90.000,B 90.000,C 0.000} C_DIS
LIN {X 80.207,Y -19.652,Z -59.587,A -90.000,B 90.000,C 0.000} C_DIS
LIN {X 80.335,Y -19.818,Z -59.662,A -90.000,B 90.000,C 0.000} C_DIS
LIN {X 80.339,Y -25.696,Z -59.664,A -90.000,B 90.000,C 0.000} C_DIS
LIN {X 80.343,Y -25.814,Z -59.666,A -90.000,B 90.000,C 0.000} C_DIS
LIN {X 80.404,Y -26.411,Z -59.699,A -90.000,B 90.000,C 0.000} C_DIS
LIN {X 80.460,Y -26.710,Z -59.727,A -90.000,B 90.000,C 0.000} C_DIS
LIN {X 80.513,Y -26.954,Z -59.750,A -90.000,B 90.000,C 0.000} C_DIS
LIN {X 80.607,Y -27.345,Z -59.783,A -90.000,B 90.000,C 0.000} C_DIS
LIN {X 80.648,Y -27.489,Z -59.792,A -90.000,B 90.000,C 0.000} C_DIS
LIN {X 80.686,Y -27.605,Z -59.797,A -90.000,B 90.000,C 0.000} C_DIS
LIN {X 80.721,Y -27.699,Z -59.798,A -90.000,B 90.000,C 0.000} C_DIS
LIN {X 80.753,Y -27.776,Z -59.794,A -90.000,B 90.000,C 0.000} C_DIS
LIN {X 80.782,Y -27.838,Z -59.786,A -90.000,B 90.000,C 0.000} C_DIS
LIN {X 80.821,Y -27.909,Z -59.766,A -90.000,B 90.000,C 0.000} C_DIS
LIN {X 80.844,Y -27.942,Z -59.747,A -90.000,B 90.000,C 0.000} C_DIS
LIN {X 80.855,Y -27.956,Z -59.736,A -90.000,B 90.000,C 0.000} C_DIS
LIN {X 80.875,Y -27.975,Z -59.710,A -90.000,B 90.000,C 0.000} C_DIS
LIN {X 80.893,Y -27.986,Z -59.681,A -90.000,B 90.000,C 0.000} C_DIS
LIN {X 80.909,Y -27.990,Z -59.647,A -90.000,B 90.000,C 0.000} C_DIS
LIN {X 80.923,Y -27.986,Z -59.609,A -90.000,B 90.000,C 0.000} C_DIS
LIN {X 80.936,Y -27.976,Z -59.566,A -90.000,B 90.000,C 0.000} C_DIS
LIN {X 80.948,Y -27.959,Z -59.520,A -90.000,B 90.000,C 0.000} C_DIS
LIN {X 80.959,Y -27.936,Z -59.469,A -90.000,B 90.000,C 0.000} C_DIS
LIN {X 80.979,Y -27.872,Z -59.356,A -90.000,B 90.000,C 0.000} C_DIS
LIN {X 80.997,Y -27.784,Z -59.226,A -90.000,B 90.000,C 0.000} C_DIS
LIN {X 81.014,Y -27.671,Z -59.081,A -90.000,B 90.000,C 0.000} C_DIS
LIN {X 81.032,Y -27.531,Z -58.919,A -90.000,B 90.000,C 0.000} C_DIS
LIN {X 81.053,Y -27.430,Z -58.743,A -90.000,B 90.000,C 0.000} C_DIS
LIN {X 81.107,Y -27.219,Z -58.344,A -90.000,B 90.000,C 0.000} C_DIS
LIN {X 81.164,Y -27.042,Z -58.006,A -90.000,B 90.000,C 0.000} C_DIS
LIN {X 81.213,Y -26.920,Z -57.762,A -90.000,B 90.000,C 0.000} C_DIS
LIN {X 81.241,Y -26.860,Z -57.635,A -90.000,B 90.000,C 0.000} C_DIS
LIN {X 81.306,Y -26.740,Z -57.370,A -90.000,B 90.000,C 0.000} C_DIS
LIN {X 81.343,Y -26.662,Z -57.233,A -90.000,B 90.000,C 0.000} C_DIS
LIN {X 81.427,Y -26.471,Z -56.947,A -90.000,B 90.000,C 0.000} C_DIS
LIN {X 81.525,Y -26.268,Z -56.648,A -90.000,B 90.000,C 0.000} C_DIS
LIN {X 81.639,Y -26.049,Z -56.335,A -90.000,B 90.000,C 0.000} C_DIS
LIN {X 81.703,Y -9.308,Z -56.174,A -90.000,B 90.000,C 0.000} C_DIS
LIN {X 81.968,Y -9.310,Z -55.519,A -90.000,B 90.000,C 0.000} C_DIS
LIN {X 81.974,Y -9.308,Z -55.505,A -90.000,B 90.000,C 0.000} C_DIS
LIN {X 81.974,Y -60.000,Z -55.505,A -90.000,B 90.000,C 0.000} C_DIS
LIN {X -120.015,Y -60.000,Z -239.406,A -90.000,B 90.000,C 0.000} C_DIS
LIN {X -120.015,Y -9.308,Z -239.406,A -90.000,B 90.000,C 0.000} C_DIS
LIN {X -117.961,Y -9.308,Z -238.027,A -90.000,B 90.000,C 0.000} C_DIS
LIN {X -116.630,Y -9.308,Z -237.143,A -90.000,B 90.000,C 0.000} C_DIS
LIN {X -110.504,Y -9.308,Z -233.086,A -90.000,B 90.000,C 0.000} C_DIS
LIN {X -109.322,Y -9.308,Z -232.312,A -90.000,B 90.000,C 0.000} C_DIS
LIN {X -102.783,Y -9.308,Z -228.042,A -90.000,B 90.000,C 0.000} C_DIS
LIN {X -100.143,Y -9.308,Z -226.346,A -90.000,B 90.000,C 0.000} C_DIS
LIN {X -94.802,Y -9.308,Z -222.919,A -90.000,B 90.000,C 0.000} C_DIS
LIN {X -86.587,Y -9.308,Z -217.763,A -90.000,B 90.000,C 0.000} C_DIS
LIN {X -83.823,Y -9.308,Z -216.070,A -90.000,B 90.000,C 0.000} C_DIS
LIN {X -78.156,Y -9.308,Z -212.620,A -90.000,B 90.000,C 0.000} C_DIS
LIN {X -76.814,Y -9.308,Z -211.809,A -90.000,B 90.000,C 0.000} C_DIS
LIN {X -70.357,Y -9.308,Z -207.946,A -90.000,B 90.000,C 0.000} C_DIS
LIN {X -61.851,Y -9.308,Z -202.906,A -90.000,B 90.000,C 0.000} C_DIS
LIN {X -55.836,Y -9.308,Z -199.328,A -90.000,B 90.000,C 0.000} C_DIS
LIN {X -54.880,Y -9.308,Z -198.766,A -90.000,B 90.000,C 0.000} C_DIS
LIN {X -53.894,Y -9.308,Z -198.163,A -90.000,B 90.000,C 0.000} C_DIS
LIN {X -49.260,Y -9.308,Z -195.302,A -90.000,B 90.000,C 0.000} C_DIS
LIN {X -44.682,Y -9.308,Z -192.342,A -90.000,B 90.000,C 0.000} C_DIS
LIN {X -44.154,Y -9.308,Z -191.986,A -90.000,B 90.000,C 0.000} C_DIS
LIN {X -40.692,Y -9.308,Z -189.631,A -90.000,B 90.000,C 0.000} C_DIS
LIN {X -40.124,Y -9.308,Z -189.230,A -90.000,B 90.000,C 0.000} C_DIS
LIN {X -37.213,Y -9.308,Z -187.156,A -90.000,B 90.000,C 0.000} C_DIS
LIN {X -34.539,Y -9.308,Z -185.186,A -90.000,B 90.000,C 0.000} C_DIS
LIN {X -34.015,Y -9.308,Z -184.803,A -90.000,B 90.000,C 0.000} C_DIS
LIN {X -31.403,Y -9.308,Z -182.791,A -90.000,B 90.000,C 0.000} C_DIS
LIN {X -29.092,Y -9.308,Z -180.900,A -90.000,B 90.000,C 0.000} C_DIS
LIN {X -28.761,Y -9.308,Z -180.632,A -90.000,B 90.000,C 0.000} C_DIS
LIN {X -26.426,Y -9.308,Z -178.572,A -90.000,B 90.000,C 0.000} C_DIS
LIN {X -24.529,Y -9.308,Z -176.734,A -90.000,B 90.000,C 0.000} C_DIS
LIN {X -24.380,Y -9.308,Z -176.570,A -90.000,B 90.000,C 0.000} C_DIS
LIN {X -22.762,Y -9.308,Z -174.810,A -90.000,B 90.000,C 0.000} C_DIS
LIN {X -21.186,Y -9.308,Z -172.849,A -90.000,B 90.000,C 0.000} C_DIS
LIN {X -20.958,Y -9.308,Z -172.513,A -90.000,B 90.000,C 0.000} C_DIS
LIN {X -19.835,Y -9.308,Z -170.893,A -90.000,B 90.000,C 0.000} C_DIS
LIN {X -18.643,Y -9.308,Z -168.884,A -90.000,B 90.000,C 0.000} C_DIS
LIN {X -18.502,Y -9.308,Z -168.639,A -90.000,B 90.000,C 0.000} C_DIS
LIN {X -17.438,Y -9.308,Z -166.541,A -90.000,B 90.000,C 0.000} C_DIS
LIN {X -16.563,Y -9.308,Z -164.471,A -90.000,B 90.000,C 0.000} C_DIS
LIN {X -16.099,Y -9.308,Z -162.956,A -90.000,B 90.000,C 0.000} C_DIS
LIN {X -15.988,Y -9.308,Z -162.081,A -90.000,B 90.000,C 0.000} C_DIS
LIN {X -16.030,Y -9.308,Z -161.604,A -90.000,B 90.000,C 0.000} C_DIS
LIN {X -16.182,Y -9.308,Z -161.112,A -90.000,B 90.000,C 0.000} C_DIS
LIN {X -16.589,Y -9.308,Z -160.232,A -90.000,B 90.000,C 0.000} C_DIS
LIN {X -16.613,Y -9.308,Z -160.173,A -90.000,B 90.000,C 0.000} C_DIS
LIN {X -17.078,Y -9.308,Z -159.264,A -90.000,B 90.000,C 0.000} C_DIS
LIN {X -17.750,Y -9.308,Z -158.191,A -90.000,B 90.000,C 0.000} C_DIS
LIN {X -18.267,Y -9.308,Z -157.512,A -90.000,B 90.000,C 0.000} C_DIS
LIN {X -18.799,Y -9.308,Z -156.811,A -90.000,B 90.000,C 0.000} C_DIS
LIN {X -18.958,Y -9.308,Z -156.638,A -90.000,B 90.000,C 0.000} C_DIS
LIN {X -20.453,Y -9.308,Z -154.950,A -90.000,B 90.000,C 0.000} C_DIS
LIN {X -20.556,Y -9.308,Z -154.850,A -90.000,B 90.000,C 0.000} C_DIS
LIN {X -22.986,Y -9.308,Z -152.393,A -90.000,B 90.000,C 0.000} C_DIS
LIN {X -23.158,Y -9.308,Z -152.224,A -90.000,B 90.000,C 0.000} C_DIS
LIN {X -26.023,Y -9.308,Z -149.306,A -90.000,B 90.000,C 0.000} C_DIS
LIN {X -26.776,Y -9.308,Z -148.495,A -90.000,B 90.000,C 0.000} C_DIS
LIN {X -29.333,Y -9.308,Z -145.678,A -90.000,B 90.000,C 0.000} C_DIS
LIN {X -29.521,Y -9.308,Z -145.462,A -90.000,B 90.000,C 0.000} C_DIS
LIN {X -29.611,Y -9.308,Z -145.354,A -90.000,B 90.000,C 0.000} C_DIS
LIN {X -30.246,Y -9.308,Z -144.564,A -90.000,B 90.000,C 0.000} C_DIS
LIN {X -32.619,Y -9.308,Z -141.544,A -90.000,B 90.000,C 0.000} C_DIS
LIN {X -32.897,Y -9.308,Z -141.145,A -90.000,B 90.000,C 0.000} C_DIS
LIN {X -34.788,Y -9.308,Z -138.098,A -90.000,B 90.000,C 0.000} C_DIS
LIN {X -35.440,Y -9.308,Z -137.065,A -90.000,B 90.000,C 0.000} C_DIS
LIN {X -35.676,Y -9.308,Z -136.639,A -90.000,B 90.000,C 0.000} C_DIS
LIN {X -37.122,Y -9.308,Z -133.847,A -90.000,B 90.000,C 0.000} C_DIS
LIN {X -37.786,Y -9.308,Z -132.574,A -90.000,B 90.000,C 0.000} C_DIS
LIN {X -39.496,Y -9.308,Z -128.807,A -90.000,B 90.000,C 0.000} C_DIS
LIN {X -40.394,Y -9.308,Z -126.685,A -90.000,B 90.000,C 0.000} C_DIS
LIN {X -41.005,Y -9.308,Z -125.223,A -90.000,B 90.000,C 0.000} C_DIS
LIN {X -41.465,Y -9.308,Z -124.148,A -90.000,B 90.000,C 0.000} C_DIS
LIN {X -41.848,Y -9.308,Z -123.270,A -90.000,B 90.000,C 0.000} C_DIS
LIN {X -42.465,Y -9.308,Z -121.980,A -90.000,B 90.000,C 0.000} C_DIS
LIN {X -42.658,Y -9.308,Z -121.585,A -90.000,B 90.000,C 0.000} C_DIS
LIN {X -43.400,Y -9.308,Z -120.312,A -90.000,B 90.000,C 0.000} C_DIS
LIN {X -44.316,Y -9.308,Z -119.008,A -90.000,B 90.000,C 0.000} C_DIS
LIN {X -44.418,Y -9.308,Z -118.876,A -90.000,B 90.000,C 0.000} C_DIS
LIN {X -45.446,Y -9.308,Z -117.568,A -90.000,B 90.000,C 0.000} C_DIS
LIN {X -45.954,Y -9.308,Z -116.919,A -90.000,B 90.000,C 0.000} C_DIS
LIN {X -47.682,Y -9.308,Z -114.796,A -90.000,B 90.000,C 0.000} C_DIS
LIN {X -47.949,Y -9.308,Z -114.474,A -90.000,B 90.000,C 0.000} C_DIS
LIN {X -49.645,Y -9.308,Z -112.398,A -90.000,B 90.000,C 0.000} C_DIS
LIN {X -50.195,Y -9.308,Z -111.736,A -90.000,B 90.000,C 0.000} C_DIS
LIN {X -51.703,Y -9.308,Z -109.848,A -90.000,B 90.000,C 0.000} C_DIS
LIN {X -52.578,Y -9.308,Z -108.762,A -90.000,B 90.000,C 0.000} C_DIS
LIN {X -53.843,Y -9.308,Z -107.095,A -90.000,B 90.000,C 0.000} C_DIS
LIN {X -54.971,Y -9.308,Z -105.615,A -90.000,B 90.000,C 0.000} C_DIS
LIN {X -56.792,Y -9.308,Z -103.171,A -90.000,B 90.000,C 0.000} C_DIS
LIN {X -57.345,Y -9.308,Z -102.438,A -90.000,B 90.000,C 0.000} C_DIS
LIN {X -59.411,Y -9.308,Z -99.724,A -90.000,B 90.000,C 0.000} C_DIS
LIN {X -59.641,Y -9.308,Z -99.420,A -90.000,B 90.000,C 0.000} C_DIS
LIN {X -61.685,Y -9.308,Z -96.911,A -90.000,B 90.000,C 0.000} C_DIS
LIN {X -61.748,Y -9.308,Z -96.835,A -90.000,B 90.000,C 0.000} C_DIS
LIN {X -63.509,Y -9.308,Z -94.930,A -90.000,B 90.000,C 0.000} C_DIS
LIN {X -63.753,Y -9.308,Z -94.664,A -90.000,B 90.000,C 0.000} C_DIS
LIN {X -65.449,Y -9.308,Z -93.054,A -90.000,B 90.000,C 0.000} C_DIS
LIN {X -65.656,Y -9.308,Z -92.854,A -90.000,B 90.000,C 0.000} C_DIS
LIN {X -66.426,Y -9.308,Z -92.209,A -90.000,B 90.000,C 0.000} C_DIS
LIN {X -67.721,Y -9.308,Z -91.123,A -90.000,B 90.000,C 0.000} C_DIS
LIN {X -69.489,Y -9.308,Z -89.787,A -90.000,B 90.000,C 0.000} C_DIS
LIN {X -69.685,Y -9.308,Z -89.634,A -90.000,B 90.000,C 0.000} C_DIS
LIN {X -71.879,Y -9.308,Z -88.102,A -90.000,B 90.000,C 0.000} C_DIS
LIN {X -73.813,Y -9.308,Z -86.827,A -90.000,B 90.000,C 0.000} C_DIS
LIN {X -75.239,Y -9.308,Z -85.918,A -90.000,B 90.000,C 0.000} C_DIS
LIN {X -77.704,Y -9.308,Z -84.364,A -90.000,B 90.000,C 0.000} C_DIS
LIN {X -78.418,Y -9.308,Z -83.901,A -90.000,B 90.000,C 0.000} C_DIS
LIN {X -79.279,Y -9.308,Z -83.337,A -90.000,B 90.000,C 0.000} C_DIS
LIN {X -79.653,Y -9.308,Z -83.088,A -90.000,B 90.000,C 0.000} C_DIS
LIN {X -80.500,Y -9.308,Z -82.513,A -90.000,B 90.000,C 0.000} C_DIS
LIN {X -81.005,Y -9.308,Z -82.164,A -90.000,B 90.000,C 0.000} C_DIS
LIN {X -81.575,Y -9.308,Z -81.750,A -90.000,B 90.000,C 0.000} C_DIS
LIN {X -82.184,Y -9.308,Z -81.298,A -90.000,B 90.000,C 0.000} C_DIS
LIN {X -82.942,Y -9.308,Z -80.699,A -90.000,B 90.000,C 0.000} C_DIS
LIN {X -83.623,Y -9.308,Z -80.155,A -90.000,B 90.000,C 0.000} C_DIS
LIN {X -84.634,Y -9.308,Z -79.289,A -90.000,B 90.000,C 0.000} C_DIS
LIN {X -85.604,Y -9.308,Z -78.437,A -90.000,B 90.000,C 0.000} C_DIS
LIN {X -86.545,Y -9.308,Z -77.628,A -90.000,B 90.000,C 0.000} C_DIS
LIN {X -87.098,Y -9.308,Z -77.189,A -90.000,B 90.000,C 0.000} C_DIS
LIN {X -87.836,Y -9.308,Z -76.681,A -90.000,B 90.000,C 0.000} C_DIS
LIN {X -88.521,Y -9.308,Z -76.272,A -90.000,B 90.000,C 0.000} C_DIS
LIN {X -89.151,Y -9.308,Z -75.940,A -90.000,B 90.000,C 0.000} C_DIS
LIN {X -89.758,Y -9.308,Z -75.657,A -90.000,B 90.000,C 0.000} C_DIS
LIN {X -90.409,Y -9.308,Z -75.386,A -90.000,B 90.000,C 0.000} C_DIS
LIN {X -90.718,Y -9.308,Z -75.276,A -90.000,B 90.000,C 0.000} C_DIS
LIN {X -90.914,Y -9.308,Z -75.225,A -90.000,B 90.000,C 0.000} C_DIS
LIN {X -91.080,Y -9.308,Z -75.187,A -90.000,B 90.000,C 0.000} C_DIS
LIN {X -91.235,Y -9.308,Z -75.159,A -90.000,B 90.000,C 0.000} C_DIS
LIN {X -91.840,Y -9.308,Z -75.090,A -90.000,B 90.000,C 0.000} C_DIS
LIN {X -92.385,Y -9.308,Z -75.064,A -90.000,B 90.000,C 0.000} C_DIS
LIN {X -92.497,Y -9.308,Z -75.056,A -90.000,B 90.000,C 0.000} C_DIS
LIN {X -93.155,Y -9.308,Z -75.038,A -90.000,B 90.000,C 0.000} C_DIS
LIN {X -93.211,Y -9.308,Z -75.041,A -90.000,B 90.000,C 0.000} C_DIS
LIN {X -93.962,Y -9.308,Z -75.007,A -90.000,B 90.000,C 0.000} C_DIS
LIN {X -94.280,Y -9.308,Z -75.014,A -90.000,B 90.000,C 0.000} C_DIS
LIN {X -94.753,Y -9.308,Z -74.991,A -90.000,B 90.000,C 0.000} C_DIS
LIN {X -95.004,Y -9.308,Z -74.969,A -90.000,B 90.000,C 0.000} C_DIS
LIN {X -95.644,Y -9.308,Z -74.947,A -90.000,B 90.000,C 0.000} C_DIS
LIN {X -95.878,Y -9.308,Z -74.924,A -90.000,B 90.000,C 0.000} C_DIS
LIN {X -96.135,Y -9.308,Z -74.884,A -90.000,B 90.000,C 0.000} C_DIS
LIN {X -97.202,Y -9.308,Z -74.737,A -90.000,B 90.000,C 0.000} C_DIS
LIN {X -97.418,Y -9.308,Z -74.703,A -90.000,B 90.000,C 0.000} C_DIS
LIN {X -97.550,Y -9.308,Z -74.674,A -90.000,B 90.000,C 0.000} C_DIS
LIN {X -97.851,Y -9.308,Z -74.593,A -90.000,B 90.000,C 0.000} C_DIS
LIN {X -99.250,Y -9.308,Z -74.207,A -90.000,B 90.000,C 0.000} C_DIS
LIN {X -99.319,Y -9.308,Z -74.182,A -90.000,B 90.000,C 0.000} C_DIS
LIN {X -99.716,Y -9.308,Z -74.025,A -90.000,B 90.000,C 0.000} C_DIS
LIN {X -99.762,Y -9.308,Z -74.002,A -90.000,B 90.000,C 0.000} C_DIS
LIN {X -101.096,Y -9.308,Z -73.410,A -90.000,B 90.000,C 0.000} C_DIS
LIN {X -101.498,Y -9.308,Z -73.197,A -90.000,B 90.000,C 0.000} C_DIS
LIN {X -101.583,Y -9.308,Z -73.140,A -90.000,B 90.000,C 0.000} C_DIS
LIN {X -102.940,Y -9.308,Z -72.260,A -90.000,B 90.000,C 0.000} C_DIS
LIN {X -103.317,Y -9.308,Z -72.004,A -90.000,B 90.000,C 0.000} C_DIS
LIN {X -103.680,Y -9.308,Z -71.696,A -90.000,B 90.000,C 0.000} C_DIS
LIN {X -104.732,Y -9.308,Z -70.835,A -90.000,B 90.000,C 0.000} C_DIS
LIN {X -105.079,Y -9.308,Z -70.539,A -90.000,B 90.000,C 0.000} C_DIS
LIN {X -105.676,Y -9.308,Z -69.926,A -90.000,B 90.000,C 0.000} C_DIS
LIN {X -106.385,Y -9.308,Z -69.232,A -90.000,B 90.000,C 0.000} C_DIS
LIN {X -106.697,Y -9.308,Z -68.901,A -90.000,B 90.000,C 0.000} C_DIS
LIN {X -107.700,Y -9.308,Z -67.704,A -90.000,B 90.000,C 0.000} C_DIS
LIN {X -107.830,Y -9.308,Z -67.555,A -90.000,B 90.000,C 0.000} C_DIS
LIN {X -108.104,Y -9.308,Z -67.191,A -90.000,B 90.000,C 0.000} C_DIS
LIN {X -108.328,Y -9.308,Z -66.882,A -90.000,B 90.000,C 0.000} C_DIS
LIN {X -109.065,Y -9.308,Z -65.889,A -90.000,B 90.000,C 0.000} C_DIS
LIN {X -110.007,Y -9.308,Z -64.409,A -90.000,B 90.000,C 0.000} C_DIS
LIN {X -110.248,Y -9.308,Z -64.017,A -90.000,B 90.000,C 0.000} C_DIS
LIN {X -110.965,Y -9.308,Z -62.723,A -90.000,B 90.000,C 0.000} C_DIS
LIN {X -111.248,Y -9.308,Z -62.146,A -90.000,B 90.000,C 0.000} C_DIS
LIN {X -111.472,Y -9.308,Z -61.669,A -90.000,B 90.000,C 0.000} C_DIS
LIN {X -111.812,Y -9.308,Z -60.936,A -90.000,B 90.000,C 0.000} C_DIS
LIN {X -112.020,Y -9.308,Z -60.403,A -90.000,B 90.000,C 0.000} C_DIS
LIN {X -112.290,Y -9.308,Z -59.690,A -90.000,B 90.000,C 0.000} C_DIS
LIN {X -112.516,Y -9.308,Z -59.068,A -90.000,B 90.000,C 0.000} C_DIS
LIN {X -112.611,Y -9.308,Z -58.786,A -90.000,B 90.000,C 0.000} C_DIS
LIN {X -112.786,Y -9.308,Z -58.222,A -90.000,B 90.000,C 0.000} C_DIS
LIN {X -112.913,Y -9.308,Z -57.803,A -90.000,B 90.000,C 0.000} C_DIS
LIN {X -113.200,Y -9.308,Z -56.807,A -90.000,B 90.000,C 0.000} C_DIS
LIN {X -113.257,Y -9.308,Z -56.589,A -90.000,B 90.000,C 0.000} C_DIS
LIN {X -113.484,Y -9.308,Z -55.787,A -90.000,B 90.000,C 0.000} C_DIS
LIN {X -113.571,Y -9.308,Z -55.460,A -90.000,B 90.000,C 0.000} C_DIS
LIN {X -113.829,Y -9.308,Z -54.686,A -90.000,B 90.000,C 0.000} C_DIS
LIN {X -114.095,Y -9.308,Z -53.955,A -90.000,B 90.000,C 0.000} C_DIS
LIN {X -114.274,Y -9.308,Z -53.426,A -90.000,B 90.000,C 0.000} C_DIS
LIN {X -114.372,Y -9.308,Z -53.144,A -90.000,B 90.000,C 0.000} C_DIS
LIN {X -114.514,Y -9.308,Z -52.711,A -90.000,B 90.000,C 0.000} C_DIS
LIN {X -114.704,Y -9.308,Z -51.986,A -90.000,B 90.000,C 0.000} C_DIS
LIN {X -114.796,Y -9.308,Z -51.548,A -90.000,B 90.000,C 0.000} C_DIS
LIN {X -114.868,Y -9.308,Z -50.902,A -90.000,B 90.000,C 0.000} C_DIS
LIN {X -114.911,Y -9.308,Z -50.449,A -90.000,B 90.000,C 0.000} C_DIS
LIN {X -114.926,Y -9.308,Z -50.112,A -90.000,B 90.000,C 0.000} C_DIS
LIN {X -114.931,Y -9.308,Z -49.917,A -90.000,B 90.000,C 0.000} C_DIS
LIN {X -115.123,Y -9.308,Z -49.494,A -90.000,B 90.000,C 0.000} C_DIS
LIN {X -115.251,Y -9.308,Z -49.194,A -90.000,B 90.000,C 0.000} C_DIS
LIN {X -115.467,Y -9.308,Z -48.647,A -90.000,B 90.000,C 0.000} C_DIS
LIN {X -115.602,Y -9.308,Z -48.260,A -90.000,B 90.000,C 0.000} C_DIS
LIN {X -115.751,Y -9.308,Z -47.782,A -90.000,B 90.000,C 0.000} C_DIS
LIN {X -115.784,Y -9.308,Z -47.668,A -90.000,B 90.000,C 0.000} C_DIS
LIN {X -115.977,Y -9.308,Z -46.835,A -90.000,B 90.000,C 0.000} C_DIS
LIN {X -116.046,Y -9.308,Z -46.341,A -90.000,B 90.000,C 0.000} C_DIS
LIN {X -116.125,Y -9.308,Z -45.517,A -90.000,B 90.000,C 0.000} C_DIS
LIN {X -116.118,Y -9.308,Z -45.030,A -90.000,B 90.000,C 0.000} C_DIS
LIN {X -116.080,Y -9.308,Z -44.541,A -90.000,B 90.000,C 0.000} C_DIS
LIN {X -116.067,Y -9.308,Z -44.327,A -90.000,B 90.000,C 0.000} C_DIS
LIN {X -116.006,Y -9.308,Z -43.890,A -90.000,B 90.000,C 0.000} C_DIS
LIN {X -115.974,Y -9.308,Z -43.748,A -90.000,B 90.000,C 0.000} C_DIS
LIN {X -115.930,Y -9.308,Z -43.539,A -90.000,B 90.000,C 0.000} C_DIS
LIN {X -115.804,Y -9.308,Z -43.050,A -90.000,B 90.000,C 0.000} C_DIS
LIN {X -115.756,Y -9.308,Z -42.876,A -90.000,B 90.000,C 0.000} C_DIS
LIN {X -115.661,Y -9.308,Z -42.590,A -90.000,B 90.000,C 0.000} C_DIS
LIN {X -115.648,Y -9.308,Z -42.544,A -90.000,B 90.000,C 0.000} C_DIS
LIN {X -115.496,Y -9.308,Z -42.148,A -90.000,B 90.000,C 0.000} C_DIS
LIN {X -115.382,Y -9.308,Z -41.879,A -90.000,B 90.000,C 0.000} C_DIS
LIN {X -115.617,Y -9.308,Z -41.326,A -90.000,B 90.000,C 0.000} C_DIS
LIN {X -115.854,Y -9.308,Z -40.726,A -90.000,B 90.000,C 0.000} C_DIS
LIN {X -116.063,Y -9.308,Z -40.151,A -90.000,B 90.000,C 0.000} C_DIS
LIN {X -116.198,Y -9.308,Z -39.751,A -90.000,B 90.000,C 0.000} C_DIS
LIN {X -116.421,Y -9.308,Z -38.944,A -90.000,B 90.000,C 0.000} C_DIS
LIN {X -116.487,Y -9.308,Z -38.626,A -90.000,B 90.000,C 0.000} C_DIS
LIN {X -116.583,Y -9.308,Z -38.079,A -90.000,B 90.000,C 0.000} C_DIS
LIN {X -116.677,Y -9.308,Z -37.307,A -90.000,B 90.000,C 0.000} C_DIS
LIN {X -116.693,Y -9.308,Z -37.003,A -90.000,B 90.000,C 0.000} C_DIS
LIN {X -116.700,Y -9.308,Z -36.536,A -90.000,B 90.000,C 0.000} C_DIS
LIN {X -116.694,Y -9.308,Z -36.213,A -90.000,B 90.000,C 0.000} C_DIS
LIN {X -116.692,Y -9.308,Z -36.165,A -90.000,B 90.000,C 0.000} C_DIS
LIN {X -116.656,Y -9.308,Z -35.780,A -90.000,B 90.000,C 0.000} C_DIS
LIN {X -116.626,Y -9.308,Z -35.478,A -90.000,B 90.000,C 0.000} C_DIS
LIN {X -116.572,Y -9.308,Z -35.075,A -90.000,B 90.000,C 0.000} C_DIS
LIN {X -116.549,Y -9.308,Z -34.945,A -90.000,B 90.000,C 0.000} C_DIS
LIN {X -116.519,Y -9.308,Z -34.792,A -90.000,B 90.000,C 0.000} C_DIS
LIN {X -116.387,Y -9.308,Z -34.240,A -90.000,B 90.000,C 0.000} C_DIS
LIN {X -116.343,Y -9.308,Z -34.072,A -90.000,B 90.000,C 0.000} C_DIS
LIN {X -116.315,Y -9.308,Z -33.981,A -90.000,B 90.000,C 0.000} C_DIS
LIN {X -116.255,Y -9.308,Z -33.800,A -90.000,B 90.000,C 0.000} C_DIS
LIN {X -116.075,Y -9.308,Z -33.296,A -90.000,B 90.000,C 0.000} C_DIS
LIN {X -116.001,Y -9.308,Z -33.103,A -90.000,B 90.000,C 0.000} C_DIS
LIN {X -115.873,Y -9.308,Z -32.802,A -90.000,B 90.000,C 0.000} C_DIS
LIN {X -115.841,Y -9.308,Z -32.731,A -90.000,B 90.000,C 0.000} C_DIS
LIN {X -115.723,Y -9.308,Z -32.487,A -90.000,B 90.000,C 0.000} C_DIS
LIN {X -115.519,Y -9.308,Z -32.088,A -90.000,B 90.000,C 0.000} C_DIS
LIN {X -115.263,Y -9.308,Z -31.675,A -90.000,B 90.000,C 0.000} C_DIS
LIN {X -115.189,Y -9.308,Z -31.559,A -90.000,B 90.000,C 0.000} C_DIS
LIN {X -115.018,Y -9.308,Z -31.309,A -90.000,B 90.000,C 0.000} C_DIS
LIN {X -114.830,Y -9.308,Z -31.066,A -90.000,B 90.000,C 0.000} C_DIS
LIN {X -114.545,Y -9.308,Z -30.730,A -90.000,B 90.000,C 0.000} C_DIS
LIN {X -114.323,Y -9.308,Z -30.499,A -90.000,B 90.000,C 0.000} C_DIS
LIN {X -114.075,Y -9.308,Z -30.261,A -90.000,B 90.000,C 0.000} C_DIS
LIN {X -113.810,Y -9.308,Z -29.998,A -90.000,B 90.000,C 0.000} C_DIS
LIN {X -113.779,Y -9.308,Z -29.961,A -90.000,B 90.000,C 0.000} C_DIS
LIN {X -113.644,Y -9.308,Z -29.775,A -90.000,B 90.000,C 0.000} C_DIS
LIN {X -113.431,Y -9.308,Z -29.451,A -90.000,B 90.000,C 0.000} C_DIS
LIN {X -113.238,Y -9.308,Z -29.156,A -90.000,B 90.000,C 0.000} C_DIS
LIN {X -112.824,Y -9.308,Z -28.540,A -90.000,B 90.000,C 0.000} C_DIS
LIN {X -112.682,Y -9.308,Z -28.336,A -90.000,B 90.000,C 0.000} C_DIS
LIN {X -112.529,Y -9.308,Z -28.140,A -90.000,B 90.000,C 0.000} C_DIS
LIN {X -112.341,Y -9.308,Z -27.891,A -90.000,B 90.000,C 0.000} C_DIS
LIN {X -111.992,Y -9.308,Z -27.482,A -90.000,B 90.000,C 0.000} C_DIS
LIN {X -111.849,Y -9.308,Z -27.317,A -90.000,B 90.000,C 0.000} C_DIS
LIN {X -111.685,Y -9.308,Z -27.124,A -90.000,B 90.000,C 0.000} C_DIS
LIN {X -111.515,Y -9.308,Z -26.949,A -90.000,B 90.000,C 0.000} C_DIS
LIN {X -111.286,Y -9.308,Z -26.709,A -90.000,B 90.000,C 0.000} C_DIS
LIN {X -110.964,Y -9.308,Z -26.407,A -90.000,B 90.000,C 0.000} C_DIS
LIN {X -110.537,Y -9.308,Z -26.012,A -90.000,B 90.000,C 0.000} C_DIS
LIN {X -110.038,Y -9.308,Z -25.605,A -90.000,B 90.000,C 0.000} C_DIS
LIN {X -109.937,Y -9.308,Z -25.525,A -90.000,B 90.000,C 0.000} C_DIS
LIN {X -109.687,Y -9.308,Z -25.348,A -90.000,B 90.000,C 0.000} C_DIS
LIN {X -109.084,Y -9.308,Z -24.938,A -90.000,B 90.000,C 0.000} C_DIS
LIN {X -108.122,Y -9.308,Z -24.418,A -90.000,B 90.000,C 0.000} C_DIS
LIN {X -107.417,Y -9.308,Z -24.122,A -90.000,B 90.000,C 0.000} C_DIS
LIN {X -107.072,Y -9.308,Z -23.984,A -90.000,B 90.000,C 0.000} C_DIS
LIN {X -107.023,Y -9.308,Z -23.966,A -90.000,B 90.000,C 0.000} C_DIS
LIN {X -106.165,Y -9.308,Z -23.690,A -90.000,B 90.000,C 0.000} C_DIS
LIN {X -105.801,Y -9.308,Z -23.582,A -90.000,B 90.000,C 0.000} C_DIS
LIN {X -105.609,Y -9.308,Z -23.533,A -90.000,B 90.000,C 0.000} C_DIS
LIN {X -104.799,Y -9.308,Z -23.319,A -90.000,B 90.000,C 0.000} C_DIS
LIN {X -104.714,Y -9.308,Z -23.302,A -90.000,B 90.000,C 0.000} C_DIS
LIN {X -104.161,Y -9.308,Z -23.180,A -90.000,B 90.000,C 0.000} C_DIS
LIN {X -103.807,Y -9.308,Z -23.104,A -90.000,B 90.000,C 0.000} C_DIS
LIN {X -103.706,Y -9.308,Z -23.081,A -90.000,B 90.000,C 0.000} C_DIS
LIN {X -103.302,Y -9.308,Z -23.005,A -90.000,B 90.000,C 0.000} C_DIS
LIN {X -102.803,Y -9.308,Z -22.918,A -90.000,B 90.000,C 0.000} C_DIS
LIN {X -102.605,Y -9.308,Z -22.878,A -90.000,B 90.000,C 0.000} C_DIS
LIN {X -102.246,Y -9.308,Z -22.810,A -90.000,B 90.000,C 0.000} C_DIS
LIN {X -102.038,Y -9.308,Z -22.773,A -90.000,B 90.000,C 0.000} C_DIS
LIN {X -101.984,Y -9.308,Z -22.652,A -90.000,B 90.000,C 0.000} C_DIS
LIN {X -101.677,Y -9.308,Z -22.088,A -90.000,B 90.000,C 0.000} C_DIS
LIN {X -101.567,Y -9.308,Z -21.926,A -90.000,B 90.000,C 0.000} C_DIS
LIN {X -101.279,Y -9.308,Z -21.509,A -90.000,B 90.000,C 0.000} C_DIS
LIN {X -101.219,Y -9.308,Z -21.433,A -90.000,B 90.000,C 0.000} C_DIS
LIN {X -100.863,Y -9.308,Z -21.016,A -90.000,B 90.000,C 0.000} C_DIS
LIN {X -100.761,Y -9.308,Z -20.910,A -90.000,B 90.000,C 0.000} C_DIS
LIN {X -100.583,Y -9.308,Z -20.730,A -90.000,B 90.000,C 0.000} C_DIS
LIN {X -100.419,Y -9.308,Z -20.575,A -90.000,B 90.000,C 0.000} C_DIS
LIN {X -100.176,Y -9.308,Z -20.372,A -90.000,B 90.000,C 0.000} C_DIS
LIN {X -99.937,Y -9.308,Z -20.177,A -90.000,B 90.000,C 0.000} C_DIS
LIN {X -99.781,Y -9.308,Z -20.060,A -90.000,B 90.000,C 0.000} C_DIS
LIN {X -99.648,Y -9.308,Z -19.968,A -90.000,B 90.000,C 0.000} C_DIS
LIN {X -99.492,Y -9.308,Z -19.857,A -90.000,B 90.000,C 0.000} C_DIS
LIN {X -99.036,Y -9.308,Z -19.558,A -90.000,B 90.000,C 0.000} C_DIS
LIN {X -98.719,Y -9.308,Z -19.354,A -90.000,B 90.000,C 0.000} C_DIS
LIN {X -98.287,Y -9.308,Z -19.044,A -90.000,B 90.000,C 0.000} C_DIS
LIN {X -97.804,Y -9.308,Z -18.694,A -90.000,B 90.000,C 0.000} C_DIS
LIN {X -97.558,Y -9.308,Z -18.508,A -90.000,B 90.000,C 0.000} C_DIS
LIN {X -97.080,Y -9.308,Z -18.161,A -90.000,B 90.000,C 0.000} C_DIS
LIN {X -96.631,Y -9.308,Z -17.846,A -90.000,B 90.000,C 0.000} C_DIS
LIN {X -96.232,Y -9.308,Z -17.584,A -90.000,B 90.000,C 0.000} C_DIS
LIN {X -95.555,Y -9.308,Z -17.176,A -90.000,B 90.000,C 0.000} C_DIS
LIN {X -95.335,Y -9.308,Z -17.062,A -90.000,B 90.000,C 0.000} C_DIS
LIN {X -94.830,Y -9.308,Z -16.815,A -90.000,B 90.000,C 0.000} C_DIS
LIN {X -94.364,Y -9.308,Z -16.591,A -90.000,B 90.000,C 0.000} C_DIS
LIN {X -93.909,Y -9.308,Z -16.428,A -90.000,B 90.000,C 0.000} C_DIS
LIN {X -93.408,Y -9.308,Z -16.266,A -90.000,B 90.000,C 0.000} C_DIS
LIN {X -93.139,Y -9.308,Z -16.173,A -90.000,B 90.000,C 0.000} C_DIS
LIN {X -92.670,Y -9.308,Z -16.057,A -90.000,B 90.000,C 0.000} C_DIS
LIN {X -91.743,Y -9.308,Z -15.862,A -90.000,B 90.000,C 0.000} C_DIS
LIN {X -91.264,Y -9.308,Z -15.796,A -90.000,B 90.000,C 0.000} C_DIS
LIN {X -90.195,Y -9.308,Z -15.674,A -90.000,B 90.000,C 0.000} C_DIS
LIN {X -89.022,Y -9.308,Z -15.629,A -90.000,B 90.000,C 0.000} C_DIS
LIN {X -88.597,Y -9.308,Z -15.619,A -90.000,B 90.000,C 0.000} C_DIS
LIN {X -88.514,Y -9.308,Z -15.616,A -90.000,B 90.000,C 0.000} C_DIS
LIN {X -88.001,Y -9.308,Z -15.593,A -90.000,B 90.000,C 0.000} C_DIS
LIN {X -87.835,Y -9.308,Z -15.548,A -90.000,B 90.000,C 0.000} C_DIS
LIN {X -87.675,Y -9.308,Z -15.487,A -90.000,B 90.000,C 0.000} C_DIS
LIN {X -87.356,Y -9.308,Z -15.377,A -90.000,B 90.000,C 0.000} C_DIS
LIN {X -87.285,Y -9.308,Z -15.343,A -90.000,B 90.000,C 0.000} C_DIS
LIN {X -86.928,Y -9.308,Z -15.183,A -90.000,B 90.000,C 0.000} C_DIS
LIN {X -86.578,Y -9.308,Z -14.989,A -90.000,B 90.000,C 0.000} C_DIS
LIN {X -86.512,Y -9.308,Z -14.949,A -90.000,B 90.000,C 0.000} C_DIS
LIN {X -86.054,Y -9.308,Z -14.687,A -90.000,B 90.000,C 0.000} C_DIS
LIN {X -85.704,Y -9.308,Z -14.494,A -90.000,B 90.000,C 0.000} C_DIS
LIN {X -85.540,Y -9.308,Z -14.410,A -90.000,B 90.000,C 0.000} C_DIS
LIN {X -85.075,Y -9.308,Z -14.196,A -90.000,B 90.000,C 0.000} C_DIS
LIN {X -84.995,Y -9.308,Z -14.162,A -90.000,B 90.000,C 0.000} C_DIS
LIN {X -84.587,Y -9.308,Z -13.973,A -90.000,B 90.000,C 0.000} C_DIS
LIN {X -84.493,Y -9.308,Z -13.936,A -90.000,B 90.000,C 0.000} C_DIS
LIN {X -84.010,Y -9.308,Z -13.772,A -90.000,B 90.000,C 0.000} C_DIS
LIN {X -83.764,Y -9.308,Z -13.704,A -90.000,B 90.000,C 0.000} C_DIS
LIN {X -83.262,Y -9.308,Z -13.533,A -90.000,B 90.000,C 0.000} C_DIS
LIN {X -82.757,Y -9.308,Z -13.417,A -90.000,B 90.000,C 0.000} C_DIS
LIN {X -82.473,Y -9.308,Z -13.366,A -90.000,B 90.000,C 0.000} C_DIS
LIN {X -82.306,Y -9.308,Z -13.325,A -90.000,B 90.000,C 0.000} C_DIS
LIN {X -81.848,Y -9.308,Z -13.220,A -90.000,B 90.000,C 0.000} C_DIS
LIN {X -81.312,Y -9.308,Z -13.151,A -90.000,B 90.000,C 0.000} C_DIS
LIN {X -81.164,Y -9.308,Z -13.135,A -90.000,B 90.000,C 0.000} C_DIS
LIN {X -80.817,Y -9.308,Z -13.081,A -90.000,B 90.000,C 0.000} C_DIS
LIN {X -80.290,Y -9.308,Z -13.015,A -90.000,B 90.000,C 0.000} C_DIS
LIN {X -80.085,Y -9.308,Z -13.002,A -90.000,B 90.000,C 0.000} C_DIS
LIN {X -79.491,Y -9.308,Z -12.990,A -90.000,B 90.000,C 0.000} C_DIS
LIN {X -79.041,Y -9.308,Z -12.977,A -90.000,B 90.000,C 0.000} C_DIS
LIN {X -78.723,Y -9.308,Z -12.970,A -90.000,B 90.000,C 0.000} C_DIS
LIN {X -78.236,Y -9.308,Z -12.997,A -90.000,B 90.000,C 0.000} C_DIS
LIN {X -77.751,Y -9.308,Z -13.036,A -90.000,B 90.000,C 0.000} C_DIS
LIN {X -77.208,Y -9.308,Z -13.098,A -90.000,B 90.000,C 0.000} C_DIS
LIN {X -76.729,Y -9.308,Z -13.188,A -90.000,B 90.000,C 0.000} C_DIS
LIN {X -76.221,Y -9.308,Z -13.315,A -90.000,B 90.000,C 0.000} C_DIS
LIN {X -75.541,Y -9.308,Z -13.471,A -90.000,B 90.000,C 0.000} C_DIS
LIN {X -75.074,Y -9.308,Z -13.609,A -90.000,B 90.000,C 0.000} C_DIS
LIN {X -74.458,Y -9.308,Z -13.822,A -90.000,B 90.000,C 0.000} C_DIS
LIN {X -74.208,Y -9.308,Z -13.916,A -90.000,B 90.000,C 0.000} C_DIS
LIN {X -74.074,Y -9.308,Z -13.960,A -90.000,B 90.000,C 0.000} C_DIS
LIN {X -73.623,Y -9.308,Z -14.146,A -90.000,B 90.000,C 0.000} C_DIS
LIN {X -73.444,Y -9.308,Z -14.224,A -90.000,B 90.000,C 0.000} C_DIS
LIN {X -72.769,Y -9.308,Z -14.480,A -90.000,B 90.000,C 0.000} C_DIS
LIN {X -72.329,Y -9.308,Z -14.661,A -90.000,B 90.000,C 0.000} C_DIS
LIN {X -71.161,Y -9.308,Z -15.150,A -90.000,B 90.000,C 0.000} C_DIS
LIN {X -70.141,Y -9.308,Z -15.585,A -90.000,B 90.000,C 0.000} C_DIS
LIN {X -69.691,Y -9.308,Z -15.770,A -90.000,B 90.000,C 0.000} C_DIS
LIN {X -68.585,Y -9.308,Z -16.249,A -90.000,B 90.000,C 0.000} C_DIS
LIN {X -68.222,Y -9.308,Z -16.398,A -90.000,B 90.000,C 0.000} C_DIS
LIN {X -67.093,Y -9.308,Z -16.891,A -90.000,B 90.000,C 0.000} C_DIS
LIN {X -66.684,Y -9.308,Z -17.061,A -90.000,B 90.000,C 0.000} C_DIS
LIN {X -66.476,Y -9.308,Z -17.151,A -90.000,B 90.000,C 0.000} C_DIS
LIN {X -66.192,Y -9.308,Z -17.149,A -90.000,B 90.000,C 0.000} C_DIS
LIN {X -65.941,Y -9.308,Z -17.167,A -90.000,B 90.000,C 0.000} C_DIS
LIN {X -65.250,Y -9.308,Z -17.198,A -90.000,B 90.000,C 0.000} C_DIS
LIN {X -64.900,Y -9.308,Z -17.226,A -90.000,B 90.000,C 0.000} C_DIS
LIN {X -64.505,Y -9.308,Z -17.260,A -90.000,B 90.000,C 0.000} C_DIS
LIN {X -64.471,Y -9.308,Z -17.263,A -90.000,B 90.000,C 0.000} C_DIS
LIN {X -63.562,Y -9.308,Z -17.384,A -90.000,B 90.000,C 0.000} C_DIS
LIN {X -63.213,Y -9.308,Z -17.425,A -90.000,B 90.000,C 0.000} C_DIS
LIN {X -62.575,Y -9.308,Z -17.514,A -90.000,B 90.000,C 0.000} C_DIS
LIN {X -62.028,Y -9.308,Z -17.584,A -90.000,B 90.000,C 0.000} C_DIS
LIN {X -61.626,Y -9.308,Z -17.624,A -90.000,B 90.000,C 0.000} C_DIS
LIN {X -61.180,Y -9.308,Z -17.665,A -90.000,B 90.000,C 0.000} C_DIS
LIN {X -60.444,Y -9.308,Z -17.673,A -90.000,B 90.000,C 0.000} C_DIS
LIN {X -60.186,Y -9.308,Z -17.680,A -90.000,B 90.000,C 0.000} C_DIS
LIN {X -59.197,Y -9.308,Z -17.671,A -90.000,B 90.000,C 0.000} C_DIS
LIN {X -58.993,Y -9.308,Z -17.672,A -90.000,B 90.000,C 0.000} C_DIS
LIN {X -57.758,Y -9.308,Z -17.734,A -90.000,B 90.000,C 0.000} C_DIS
LIN {X -56.548,Y -9.308,Z -17.843,A -90.000,B 90.000,C 0.000} C_DIS
LIN {X -55.504,Y -9.308,Z -17.997,A -90.000,B 90.000,C 0.000} C_DIS
LIN {X -54.722,Y -9.308,Z -18.121,A -90.000,B 90.000,C 0.000} C_DIS
LIN {X -53.004,Y -9.308,Z -18.443,A -90.000,B 90.000,C 0.000} C_DIS
LIN {X -50.924,Y -9.308,Z -18.862,A -90.000,B 90.000,C 0.000} C_DIS
LIN {X -49.598,Y -9.308,Z -19.135,A -90.000,B 90.000,C 0.000} C_DIS
LIN {X -48.006,Y -9.308,Z -19.483,A -90.000,B 90.000,C 0.000} C_DIS
LIN {X -45.480,Y -9.308,Z -20.050,A -90.000,B 90.000,C 0.000} C_DIS
LIN {X -45.054,Y -9.308,Z -20.144,A -90.000,B 90.000,C 0.000} C_DIS
LIN {X -44.825,Y -9.308,Z -20.194,A -90.000,B 90.000,C 0.000} C_DIS
LIN {X -44.050,Y -9.308,Z -20.369,A -90.000,B 90.000,C 0.000} C_DIS
LIN {X -42.136,Y -9.308,Z -20.751,A -90.000,B 90.000,C 0.000} C_DIS
LIN {X -39.180,Y -9.308,Z -21.363,A -90.000,B 90.000,C 0.000} C_DIS
LIN {X -38.076,Y -9.308,Z -21.618,A -90.000,B 90.000,C 0.000} C_DIS
LIN {X -37.561,Y -9.308,Z -21.725,A -90.000,B 90.000,C 0.000} C_DIS
LIN {X -34.749,Y -9.308,Z -22.353,A -90.000,B 90.000,C 0.000} C_DIS
LIN {X -33.138,Y -9.308,Z -22.689,A -90.000,B 90.000,C 0.000} C_DIS
LIN {X -31.815,Y -9.308,Z -22.981,A -90.000,B 90.000,C 0.000} C_DIS
LIN {X -29.666,Y -9.308,Z -23.440,A -90.000,B 90.000,C 0.000} C_DIS
LIN {X -26.870,Y -9.308,Z -24.053,A -90.000,B 90.000,C 0.000} C_DIS
LIN {X -22.326,Y -9.308,Z -25.112,A -90.000,B 90.000,C 0.000} C_DIS
LIN {X -20.512,Y -9.308,Z -25.533,A -90.000,B 90.000,C 0.000} C_DIS
LIN {X -19.740,Y -9.308,Z -25.708,A -90.000,B 90.000,C 0.000} C_DIS
LIN {X -18.383,Y -9.308,Z -26.022,A -90.000,B 90.000,C 0.000} C_DIS
LIN {X -17.300,Y -9.308,Z -26.267,A -90.000,B 90.000,C 0.000} C_DIS
LIN {X -16.185,Y -9.308,Z -26.524,A -90.000,B 90.000,C 0.000} C_DIS
LIN {X -14.709,Y -9.308,Z -26.858,A -90.000,B 90.000,C 0.000} C_DIS
LIN {X -11.900,Y -9.308,Z -27.494,A -90.000,B 90.000,C 0.000} C_DIS
LIN {X -8.927,Y -9.308,Z -28.151,A -90.000,B 90.000,C 0.000} C_DIS
LIN {X -5.942,Y -9.308,Z -28.793,A -90.000,B 90.000,C 0.000} C_DIS
LIN {X -5.661,Y -9.308,Z -28.856,A -90.000,B 90.000,C 0.000} C_DIS
LIN {X -2.894,Y -9.308,Z -29.441,A -90.000,B 90.000,C 0.000} C_DIS
LIN {X -1.134,Y -9.308,Z -29.777,A -90.000,B 90.000,C 0.000} C_DIS
LIN {X 1.277,Y -9.308,Z -30.213,A -90.000,B 90.000,C 0.000} C_DIS
LIN {X 2.767,Y -9.308,Z -30.457,A -90.000,B 90.000,C 0.000} C_DIS
LIN {X 3.663,Y -9.308,Z -30.621,A -90.000,B 90.000,C 0.000} C_DIS
LIN {X 5.504,Y -9.308,Z -30.913,A -90.000,B 90.000,C 0.000} C_DIS
LIN {X 5.941,Y -9.308,Z -31.001,A -90.000,B 90.000,C 0.000} C_DIS
LIN {X 8.072,Y -9.308,Z -31.365,A -90.000,B 90.000,C 0.000} C_DIS
LIN {X 8.436,Y -9.308,Z -31.438,A -90.000,B 90.000,C 0.000} C_DIS
LIN {X 9.092,Y -9.308,Z -31.577,A -90.000,B 90.000,C 0.000} C_DIS
LIN {X 10.617,Y -9.308,Z -31.926,A -90.000,B 90.000,C 0.000} C_DIS
LIN {X 10.908,Y -9.308,Z -31.989,A -90.000,B 90.000,C 0.000} C_DIS
LIN {X 12.650,Y -9.308,Z -32.412,A -90.000,B 90.000,C 0.000} C_DIS
LIN {X 13.068,Y -9.308,Z -32.498,A -90.000,B 90.000,C 0.000} C_DIS
LIN {X 14.230,Y -9.308,Z -32.767,A -90.000,B 90.000,C 0.000} C_DIS
LIN {X 14.719,Y -9.308,Z -32.855,A -90.000,B 90.000,C 0.000} C_DIS
LIN {X 15.642,Y -9.308,Z -33.028,A -90.000,B 90.000,C 0.000} C_DIS
LIN {X 16.299,Y -9.308,Z -33.113,A -90.000,B 90.000,C 0.000} C_DIS
LIN {X 17.627,Y -9.308,Z -33.248,A -90.000,B 90.000,C 0.000} C_DIS
LIN {X 18.393,Y -9.308,Z -33.281,A -90.000,B 90.000,C 0.000} C_DIS
LIN {X 18.828,Y -9.308,Z -33.317,A -90.000,B 90.000,C 0.000} C_DIS
LIN {X 19.674,Y -9.308,Z -33.327,A -90.000,B 90.000,C 0.000} C_DIS
LIN {X 20.117,Y -9.308,Z -33.336,A -90.000,B 90.000,C 0.000} C_DIS
LIN {X 20.246,Y -9.308,Z -33.347,A -90.000,B 90.000,C 0.000} C_DIS
LIN {X 21.352,Y -9.308,Z -33.367,A -90.000,B 90.000,C 0.000} C_DIS
LIN {X 21.678,Y -9.308,Z -33.383,A -90.000,B 90.000,C 0.000} C_DIS
LIN {X 23.125,Y -9.308,Z -33.479,A -90.000,B 90.000,C 0.000} C_DIS
LIN {X 24.306,Y -9.308,Z -33.624,A -90.000,B 90.000,C 0.000} C_DIS
LIN {X 24.577,Y -9.308,Z -33.660,A -90.000,B 90.000,C 0.000} C_DIS
LIN {X 24.821,Y -9.308,Z -33.698,A -90.000,B 90.000,C 0.000} C_DIS
LIN {X 26.031,Y -9.308,Z -33.899,A -90.000,B 90.000,C 0.000} C_DIS
LIN {X 26.556,Y -9.308,Z -33.991,A -90.000,B 90.000,C 0.000} C_DIS
LIN {X 27.696,Y -9.308,Z -34.220,A -90.000,B 90.000,C 0.000} C_DIS
LIN {X 28.116,Y -9.308,Z -34.309,A -90.000,B 90.000,C 0.000} C_DIS
LIN {X 29.020,Y -9.308,Z -34.520,A -90.000,B 90.000,C 0.000} C_DIS
LIN {X 29.834,Y -9.308,Z -34.704,A -90.000,B 90.000,C 0.000} C_DIS
LIN {X 31.404,Y -9.308,Z -35.101,A -90.000,B 90.000,C 0.000} C_DIS
LIN {X 31.739,Y -9.308,Z -35.190,A -90.000,B 90.000,C 0.000} C_DIS
LIN {X 33.431,Y -9.308,Z -35.652,A -90.000,B 90.000,C 0.000} C_DIS
LIN {X 33.898,Y -9.308,Z -35.790,A -90.000,B 90.000,C 0.000} C_DIS
LIN {X 34.308,Y -9.308,Z -35.913,A -90.000,B 90.000,C 0.000} C_DIS
LIN {X 35.852,Y -9.308,Z -36.387,A -90.000,B 90.000,C 0.000} C_DIS
LIN {X 36.611,Y -9.308,Z -36.630,A -90.000,B 90.000,C 0.000} C_DIS
LIN {X 39.018,Y -9.308,Z -37.408,A -90.000,B 90.000,C 0.000} C_DIS
LIN {X 39.464,Y -9.308,Z -37.560,A -90.000,B 90.000,C 0.000} C_DIS
LIN {X 41.425,Y -9.308,Z -38.147,A -90.000,B 90.000,C 0.000} C_DIS
LIN {X 42.646,Y -9.308,Z -38.553,A -90.000,B 90.000,C 0.000} C_DIS
LIN {X 43.430,Y -9.308,Z -38.780,A -90.000,B 90.000,C 0.000} C_DIS
LIN {X 43.897,Y -9.308,Z -38.920,A -90.000,B 90.000,C 0.000} C_DIS
LIN {X 46.609,Y -9.308,Z -39.873,A -90.000,B 90.000,C 0.000} C_DIS
LIN {X 47.060,Y -9.308,Z -40.059,A -90.000,B 90.000,C 0.000} C_DIS
LIN {X 49.499,Y -9.308,Z -41.121,A -90.000,B 90.000,C 0.000} C_DIS
LIN {X 49.716,Y -9.308,Z -41.231,A -90.000,B 90.000,C 0.000} C_DIS
LIN {X 52.103,Y -9.308,Z -42.498,A -90.000,B 90.000,C 0.000} C_DIS
LIN {X 52.504,Y -9.308,Z -42.715,A -90.000,B 90.000,C 0.000} C_DIS
LIN {X 52.710,Y -9.308,Z -42.831,A -90.000,B 90.000,C 0.000} C_DIS
LIN {X 55.131,Y -9.308,Z -44.358,A -90.000,B 90.000,C 0.000} C_DIS
LIN {X 55.508,Y -9.308,Z -44.614,A -90.000,B 90.000,C 0.000} C_DIS
LIN {X 57.720,Y -9.308,Z -46.256,A -90.000,B 90.000,C 0.000} C_DIS
LIN {X 58.412,Y -9.308,Z -46.839,A -90.000,B 90.000,C 0.000} C_DIS
LIN {X 58.603,Y -9.308,Z -46.947,A -90.000,B 90.000,C 0.000} C_DIS
LIN {X 60.152,Y -9.308,Z -47.686,A -90.000,B 90.000,C 0.000} C_DIS
LIN {X 60.580,Y -9.308,Z -47.910,A -90.000,B 90.000,C 0.000} C_DIS
LIN {X 61.496,Y -9.308,Z -48.410,A -90.000,B 90.000,C 0.000} C_DIS
LIN {X 62.940,Y -9.308,Z -49.101,A -90.000,B 90.000,C 0.000} C_DIS
LIN {X 64.205,Y -9.308,Z -49.733,A -90.000,B 90.000,C 0.000} C_DIS
LIN {X 65.274,Y -9.308,Z -50.263,A -90.000,B 90.000,C 0.000} C_DIS
LIN {X 65.922,Y -9.308,Z -50.593,A -90.000,B 90.000,C 0.000} C_DIS
LIN {X 66.728,Y -9.308,Z -51.017,A -90.000,B 90.000,C 0.000} C_DIS
LIN {X 67.840,Y -9.308,Z -51.612,A -90.000,B 90.000,C 0.000} C_DIS
LIN {X 68.049,Y -9.308,Z -51.729,A -90.000,B 90.000,C 0.000} C_DIS
LIN {X 69.523,Y -9.308,Z -52.578,A -90.000,B 90.000,C 0.000} C_DIS
LIN {X 70.726,Y -9.308,Z -53.307,A -90.000,B 90.000,C 0.000} C_DIS
LIN {X 71.385,Y -9.308,Z -53.704,A -90.000,B 90.000,C 0.000} C_DIS
LIN {X 73.495,Y -9.308,Z -55.028,A -90.000,B 90.000,C 0.000} C_DIS
LIN {X 75.596,Y -9.308,Z -56.393,A -90.000,B 90.000,C 0.000} C_DIS
LIN {X 76.205,Y -9.308,Z -56.800,A -90.000,B 90.000,C 0.000} C_DIS
LIN {X 77.830,Y -9.308,Z -57.896,A -90.000,B 90.000,C 0.000} C_DIS
LIN {X 77.976,Y -9.308,Z -57.997,A -90.000,B 90.000,C 0.000} C_DIS
LIN {X 78.988,Y -9.308,Z -58.724,A -90.000,B 90.000,C 0.000} C_DIS
LIN {X 79.439,Y -9.314,Z -59.048,A -90.000,B 90.000,C 0.000} C_DIS
LIN {X 79.631,Y -9.308,Z -59.185,A -90.000,B 90.000,C 0.000} C_DIS
LIN {X 79.833,Y -9.308,Z -59.325,A -90.000,B 90.000,C 0.000} C_DIS
LIN {X 79.834,Y -17.866,Z -59.326,A -90.000,B 90.000,C 0.000} C_DIS
LIN {X 79.837,Y -17.991,Z -59.328,A -90.000,B 90.000,C 0.000} C_DIS
LIN {X 79.882,Y -18.629,Z -59.358,A -90.000,B 90.000,C 0.000} C_DIS
LIN {X 79.956,Y -19.068,Z -59.408,A -90.000,B 90.000,C 0.000} C_DIS
LIN {X 80.026,Y -19.321,Z -59.454,A -90.000,B 90.000,C 0.000} C_DIS
LIN {X 80.091,Y -19.468,Z -59.495,A -90.000,B 90.000,C 0.000} C_DIS
LIN {X 80.210,Y -19.646,Z -59.567,A -90.000,B 90.000,C 0.000} C_DIS
LIN {X 80.337,Y -19.811,Z -59.634,A -90.000,B 90.000,C 0.000} C_DIS
LIN {X 80.348,Y -25.742,Z -59.639,A -90.000,B 90.000,C 0.000} C_DIS
LIN {X 80.351,Y -25.815,Z -59.640,A -90.000,B 90.000,C 0.000} C_DIS
LIN {X 80.359,Y -25.956,Z -59.644,A -90.000,B 90.000,C 0.000} C_DIS
LIN {X 80.402,Y -26.339,Z -59.662,A -90.000,B 90.000,C 0.000} C_DIS
LIN {X 80.442,Y -26.564,Z -59.676,A -90.000,B 90.000,C 0.000} C_DIS
LIN {X 80.513,Y -26.876,Z -59.692,A -90.000,B 90.000,C 0.000} C_DIS
LIN {X 80.544,Y -26.998,Z -59.695,A -90.000,B 90.000,C 0.000} C_DIS
LIN {X 80.572,Y -27.102,Z -59.693,A -90.000,B 90.000,C 0.000} C_DIS
LIN {X 80.611,Y -27.227,Z -59.684,A -90.000,B 90.000,C 0.000} C_DIS
LIN {X 80.644,Y -27.319,Z -59.667,A -90.000,B 90.000,C 0.000} C_DIS
LIN {X 80.664,Y -27.363,Z -59.650,A -90.000,B 90.000,C 0.000} C_DIS
LIN {X 80.682,Y -27.395,Z -59.630,A -90.000,B 90.000,C 0.000} C_DIS
LIN {X 80.699,Y -27.416,Z -59.607,A -90.000,B 90.000,C 0.000} C_DIS
LIN {X 80.714,Y -27.426,Z -59.579,A -90.000,B 90.000,C 0.000} C_DIS
LIN {X 80.728,Y -27.428,Z -59.548,A -90.000,B 90.000,C 0.000} C_DIS
LIN {X 80.741,Y -27.421,Z -59.514,A -90.000,B 90.000,C 0.000} C_DIS
LIN {X 80.752,Y -27.407,Z -59.476,A -90.000,B 90.000,C 0.000} C_DIS
LIN {X 80.763,Y -27.384,Z -59.434,A -90.000,B 90.000,C 0.000} C_DIS
LIN {X 80.783,Y -27.319,Z -59.340,A -90.000,B 90.000,C 0.000} C_DIS
LIN {X 80.802,Y -27.237,Z -59.232,A -90.000,B 90.000,C 0.000} C_DIS
LIN {X 80.821,Y -27.173,Z -59.110,A -90.000,B 90.000,C 0.000} C_DIS
LIN {X 80.863,Y -27.006,Z -58.825,A -90.000,B 90.000,C 0.000} C_DIS
LIN {X 80.889,Y -26.905,Z -58.663,A -90.000,B 90.000,C 0.000} C_DIS
LIN {X 80.938,Y -26.737,Z -58.395,A -90.000,B 90.000,C 0.000} C_DIS
LIN {X 81.002,Y -26.555,Z -58.098,A -90.000,B 90.000,C 0.000} C_DIS
LIN {X 81.055,Y -26.434,Z -57.885,A -90.000,B 90.000,C 0.000} C_DIS
LIN {X 81.086,Y -26.376,Z -57.773,A -90.000,B 90.000,C 0.000} C_DIS
LIN {X 81.119,Y -26.324,Z -57.658,A -90.000,B 90.000,C 0.000} C_DIS
LIN {X 81.155,Y -26.278,Z -57.541,A -90.000,B 90.000,C 0.000} C_DIS
LIN {X 81.236,Y -26.201,Z -57.296,A -90.000,B 90.000,C 0.000} C_DIS
LIN {X 81.281,Y -26.140,Z -57.169,A -90.000,B 90.000,C 0.000} C_DIS
LIN {X 81.343,Y -26.039,Z -57.007,A -90.000,B 90.000,C 0.000} C_DIS
LIN {X 81.383,Y -25.984,Z -56.907,A -90.000,B 90.000,C 0.000} C_DIS
LIN {X 81.439,Y -25.926,Z -56.771,A -90.000,B 90.000,C 0.000} C_DIS
LIN {X 81.499,Y -9.308,Z -56.633,A -90.000,B 90.000,C 0.000} C_DIS
LIN {X 81.700,Y -9.308,Z -56.182,A -90.000,B 90.000,C 0.000} C_DIS
LIN {X 82.134,Y -9.308,Z -55.110,A -90.000,B 90.000,C 0.000} C_DIS
LIN {X 82.335,Y -9.308,Z -54.666,A -90.000,B 90.000,C 0.000} C_DIS
LIN {X 83.331,Y -9.308,Z -52.811,A -90.000,B 90.000,C 0.000} C_DIS
LIN {X 83.577,Y -9.308,Z -52.389,A -90.000,B 90.000,C 0.000} C_DIS
LIN {X 84.737,Y -9.308,Z -50.685,A -90.000,B 90.000,C 0.000} C_DIS
LIN {X 85.025,Y -9.308,Z -50.291,A -90.000,B 90.000,C 0.000} C_DIS
LIN {X 86.337,Y -9.308,Z -48.714,A -90.000,B 90.000,C 0.000} C_DIS
LIN {X 86.664,Y -9.308,Z -48.352,A -90.000,B 90.000,C 0.000} C_DIS
LIN {X 88.117,Y -9.308,Z -46.880,A -90.000,B 90.000,C 0.000} C_DIS
LIN {X 88.479,Y -9.308,Z -46.553,A -90.000,B 90.000,C 0.000} C_DIS
LIN {X 90.061,Y -9.308,Z -45.164,A -90.000,B 90.000,C 0.000} C_DIS
LIN {X 91.716,Y -9.308,Z -43.876,A -90.000,B 90.000,C 0.000} C_DIS
LIN {X 92.110,Y -9.308,Z -43.588,A -90.000,B 90.000,C 0.000} C_DIS
LIN {X 93.780,Y -9.308,Z -42.419,A -90.000,B 90.000,C 0.000} C_DIS
LIN {X 95.417,Y -9.308,Z -41.383,A -90.000,B 90.000,C 0.000} C_DIS
LIN {X 95.838,Y -9.308,Z -41.136,A -90.000,B 90.000,C 0.000} C_DIS
LIN {X 97.264,Y -9.308,Z -40.323,A -90.000,B 90.000,C 0.000} C_DIS
LIN {X 97.264,Y -60.000,Z -40.323,A -90.000,B 90.000,C 0.000} C_DIS
LIN {X 102.562,Y -60.000,Z -88.725,A -90.000,B 90.000,C 0.000} C_DIS
LIN {X 102.562,Y -9.308,Z -88.725,A -90.000,B 90.000,C 0.000} C_DIS
LIN {X 102.900,Y -9.308,Z -89.366,A -90.000,B 90.000,C 0.000} C_DIS
LIN {X 103.074,Y -9.308,Z -89.699,A -90.000,B 90.000,C 0.000} C_DIS
LIN {X 103.184,Y -9.308,Z -89.932,A -90.000,B 90.000,C 0.000} C_DIS
LIN {X 103.639,Y -9.308,Z -90.920,A -90.000,B 90.000,C 0.000} C_DIS
LIN {X 103.810,Y -9.308,Z -91.355,A -90.000,B 90.000,C 0.000} C_DIS
LIN {X 104.152,Y -9.308,Z -92.239,A -90.000,B 90.000,C 0.000} C_DIS
LIN {X 104.248,Y -9.308,Z -92.485,A -90.000,B 90.000,C 0.000} C_DIS
LIN {X 104.521,Y -9.308,Z -93.348,A -90.000,B 90.000,C 0.000} C_DIS
LIN {X 104.594,Y -9.308,Z -93.572,A -90.000,B 90.000,C 0.000} C_DIS
LIN {X 104.718,Y -9.308,Z -94.023,A -90.000,B 90.000,C 0.000} C_DIS
LIN {X 104.933,Y -9.308,Z -94.845,A -90.000,B 90.000,C 0.000} C_DIS
LIN {X 105.006,Y -9.308,Z -95.114,A -90.000,B 90.000,C 0.000} C_DIS
LIN {X 105.190,Y -9.308,Z -95.918,A -90.000,B 90.000,C 0.000} C_DIS
LIN {X 105.270,Y -9.308,Z -96.256,A -90.000,B 90.000,C 0.000} C_DIS
LIN {X 105.543,Y -9.308,Z -97.491,A -90.000,B 90.000,C 0.000} C_DIS
LIN {X 105.837,Y -9.308,Z -98.874,A -90.000,B 90.000,C 0.000} C_DIS
LIN {X 105.987,Y -9.308,Z -99.610,A -90.000,B 90.000,C 0.000} C_DIS
LIN {X 106.164,Y -9.308,Z -100.461,A -90.000,B 90.000,C 0.000} C_DIS
LIN {X 106.356,Y -9.308,Z -101.432,A -90.000,B 90.000,C 0.000} C_DIS
LIN {X 106.733,Y -9.308,Z -103.265,A -90.000,B 90.000,C 0.000} C_DIS
LIN {X 106.970,Y -9.308,Z -104.490,A -90.000,B 90.000,C 0.000} C_DIS
LIN {X 107.167,Y -9.308,Z -105.481,A -90.000,B 90.000,C 0.000} C_DIS
LIN {X 107.623,Y -9.308,Z -107.930,A -90.000,B 90.000,C 0.000} C_DIS
LIN {X 107.910,Y -9.308,Z -109.562,A -90.000,B 90.000,C 0.000} C_DIS
LIN {X 108.243,Y -9.308,Z -111.509,A -90.000,B 90.000,C 0.000} C_DIS
LIN {X 108.447,Y -9.308,Z -112.772,A -90.000,B 90.000,C 0.000} C_DIS
LIN {X 108.604,Y -9.308,Z -113.871,A -90.000,B 90.000,C 0.000} C_DIS
LIN {X 108.863,Y -9.308,Z -115.598,A -90.000,B 90.000,C 0.000} C_DIS
LIN {X 109.020,Y -9.308,Z -116.854,A -90.000,B 90.000,C 0.000} C_DIS
LIN {X 109.228,Y -9.308,Z -118.438,A -90.000,B 90.000,C 0.000} C_DIS
LIN {X 109.384,Y -9.308,Z -119.862,A -90.000,B 90.000,C 0.000} C_DIS
LIN {X 109.542,Y -9.308,Z -121.241,A -90.000,B 90.000,C 0.000} C_DIS
LIN {X 109.690,Y -9.308,Z -122.816,A -90.000,B 90.000,C 0.000} C_DIS
LIN {X 109.802,Y -9.308,Z -123.960,A -90.000,B 90.000,C 0.000} C_DIS
LIN {X 109.934,Y -9.308,Z -125.639,A -90.000,B 90.000,C 0.000} C_DIS
LIN {X 110.009,Y -9.308,Z -126.551,A -90.000,B 90.000,C 0.000} C_DIS
LIN {X 110.118,Y -9.308,Z -128.374,A -90.000,B 90.000,C 0.000} C_DIS
LIN {X 110.164,Y -9.308,Z -129.118,A -90.000,B 90.000,C 0.000} C_DIS
LIN {X 110.189,Y -9.308,Z -129.573,A -90.000,B 90.000,C 0.000} C_DIS
LIN {X 110.294,Y -9.308,Z -132.218,A -90.000,B 90.000,C 0.000} C_DIS
LIN {X 110.351,Y -9.308,Z -135.045,A -90.000,B 90.000,C 0.000} C_DIS
LIN {X 110.362,Y -9.308,Z -138.156,A -90.000,B 90.000,C 0.000} C_DIS
LIN {X 110.319,Y -9.308,Z -141.617,A -90.000,B 90.000,C 0.000} C_DIS
LIN {X 110.219,Y -9.308,Z -145.166,A -90.000,B 90.000,C 0.000} C_DIS
LIN {X 110.054,Y -9.308,Z -148.870,A -90.000,B 90.000,C 0.000} C_DIS
LIN {X 109.817,Y -9.308,Z -152.686,A -90.000,B 90.000,C 0.000} C_DIS
LIN {X 109.746,Y -9.308,Z -153.756,A -90.000,B 90.000,C 0.000} C_DIS
LIN {X 109.462,Y -9.308,Z -157.497,A -90.000,B 90.000,C 0.000} C_DIS
LIN {X 109.203,Y -9.308,Z -160.498,A -90.000,B 90.000,C 0.000} C_DIS
LIN {X 109.141,Y -9.308,Z -161.256,A -90.000,B 90.000,C 0.000} C_DIS
LIN {X 108.849,Y -9.308,Z -164.376,A -90.000,B 90.000,C 0.000} C_DIS
LIN {X 108.531,Y -9.308,Z -167.654,A -90.000,B 90.000,C 0.000} C_DIS
LIN {X 108.484,Y -9.308,Z -168.186,A -90.000,B 90.000,C 0.000} C_DIS
LIN {X 108.151,Y -9.308,Z -171.446,A -90.000,B 90.000,C 0.000} C_DIS
LIN {X 108.112,Y -9.308,Z -171.865,A -90.000,B 90.000,C 0.000} C_DIS
LIN {X 108.066,Y -9.308,Z -172.304,A -90.000,B 90.000,C 0.000} C_DIS
LIN {X 107.736,Y -9.308,Z -175.355,A -90.000,B 90.000,C 0.000} C_DIS
LIN {X 107.688,Y -9.308,Z -175.810,A -90.000,B 90.000,C 0.000} C_DIS
LIN {X 107.429,Y -9.308,Z -178.026,A -90.000,B 90.000,C 0.000} C_DIS
LIN {X 107.326,Y -9.308,Z -178.978,A -90.000,B 90.000,C 0.000} C_DIS
LIN {X 107.202,Y -9.308,Z -180.014,A -90.000,B 90.000,C 0.000} C_DIS
LIN {X 106.957,Y -9.308,Z -181.929,A -90.000,B 90.000,C 0.000} C_DIS
LIN {X 106.834,Y -9.308,Z -182.865,A -90.000,B 90.000,C 0.000} C_DIS
LIN {X 106.466,Y -9.308,Z -185.506,A -90.000,B 90.000,C 0.000} C_DIS
LIN {X 106.098,Y -9.308,Z -187.994,A -90.000,B 90.000,C 0.000} C_DIS
LIN {X 105.730,Y -9.308,Z -190.391,A -90.000,B 90.000,C 0.000} C_DIS
LIN {X 105.350,Y -9.308,Z -192.803,A -90.000,B 90.000,C 0.000} C_DIS
LIN {X 105.059,Y -9.308,Z -194.581,A -90.000,B 90.000,C 0.000} C_DIS
LIN {X 104.918,Y -9.308,Z -195.432,A -90.000,B 90.000,C 0.000} C_DIS
LIN {X 104.400,Y -9.308,Z -198.467,A -90.000,B 90.000,C 0.000} C_DIS
LIN {X 103.761,Y -9.308,Z -202.084,A -90.000,B 90.000,C 0.000} C_DIS
LIN {X 103.120,Y -9.308,Z -205.608,A -90.000,B 90.000,C 0.000} C_DIS
LIN {X 102.974,Y -9.308,Z -206.379,A -90.000,B 90.000,C 0.000} C_DIS
LIN {X 102.145,Y -9.308,Z -210.669,A -90.000,B 90.000,C 0.000} C_DIS
LIN {X 101.955,Y -9.308,Z -211.586,A -90.000,B 90.000,C 0.000} C_DIS
LIN {X 100.914,Y -9.308,Z -216.543,A -90.000,B 90.000,C 0.000} C_DIS
LIN {X 99.604,Y -9.308,Z -222.162,A -90.000,B 90.000,C 0.000} C_DIS
LIN {X 98.096,Y -9.308,Z -227.862,A -90.000,B 90.000,C 0.000} C_DIS
LIN {X 96.401,Y -9.308,Z -233.602,A -90.000,B 90.000,C 0.000} C_DIS
LIN {X 96.116,Y -9.308,Z -234.495,A -90.000,B 90.000,C 0.000} C_DIS
LIN {X 94.503,Y -9.308,Z -239.478,A -90.000,B 90.000,C 0.000} C_DIS
LIN {X 93.872,Y -9.308,Z -241.348,A -90.000,B 90.000,C 0.000} C_DIS
LIN {X 93.102,Y -9.308,Z -243.561,A -90.000,B 90.000,C 0.000} C_DIS
LIN {X 93.102,Y -60.000,Z -243.561,A -90.000,B 90.000,C 0.000} C_DIS
LIN {X -120.015,Y -60.000,Z -238.278,A -90.000,B 90.000,C 0.000} C_DIS
LIN {X -120.015,Y -7.308,Z -238.278,A -90.000,B 90.000,C 0.000} C_DIS
LIN {X -118.521,Y -7.308,Z -237.277,A -90.000,B 90.000,C 0.000} C_DIS
LIN {X -117.316,Y -7.308,Z -236.477,A -90.000,B 90.000,C 0.000} C_DIS
LIN {X -111.200,Y -7.308,Z -232.445,A -90.000,B 90.000,C 0.000} C_DIS
LIN {X -110.997,Y -7.308,Z -232.312,A -90.000,B 90.000,C 0.000} C_DIS
LIN {X -104.652,Y -7.308,Z -228.188,A -90.000,B 90.000,C 0.000} C_DIS
LIN {X -103.182,Y -7.308,Z -227.234,A -90.000,B 90.000,C 0.000} C_DIS
LIN {X -102.957,Y -7.308,Z -227.090,A -90.000,B 90.000,C 0.000} C_DIS
LIN {X -95.176,Y -7.308,Z -222.139,A -90.000,B 90.000,C 0.000} C_DIS
LIN {X -93.612,Y -7.308,Z -221.170,A -90.000,B 90.000,C 0.000} C_DIS
LIN {X -86.920,Y -7.308,Z -217.019,A -90.000,B 90.000,C 0.000} C_DIS
LIN {X -82.052,Y -7.308,Z -214.092,A -90.000,B 90.000,C 0.000} C_DIS
LIN {X -78.427,Y -7.308,Z -211.927,A -90.000,B 90.000,C 0.000} C_DIS
LIN {X -74.942,Y -7.308,Z -209.869,A -90.000,B 90.000,C 0.000} C_DIS
LIN {X -70.057,Y -7.308,Z -207.014,A -90.000,B 90.000,C 0.000} C_DIS
LIN {X -68.000,Y -7.308,Z -205.805,A -90.000,B 90.000,C 0.000} C_DIS
LIN {X -62.177,Y -7.308,Z -202.425,A -90.000,B 90.000,C 0.000} C_DIS
LIN {X -61.361,Y -7.308,Z -201.940,A -90.000,B 90.000,C 0.000} C_DIS
LIN {X -55.540,Y -7.308,Z -198.522,A -90.000,B 90.000,C 0.000} C_DIS
LIN {X -55.161,Y -7.308,Z -198.300,A -90.000,B 90.000,C 0.000} C_DIS
LIN {X -54.780,Y -7.308,Z -198.067,A -90.000,B 90.000,C 0.000} C_DIS
LIN {X -54.759,Y -7.308,Z -198.054,A -90.000,B 90.000,C 0.000} C_DIS
LIN {X -49.566,Y -7.308,Z -194.882,A -90.000,B 90.000,C 0.000} C_DIS
LIN {X -46.456,Y -7.308,Z -192.888,A -90.000,B 90.000,C 0.000} C_DIS
LIN {X -45.188,Y -7.308,Z -192.075,A -90.000,B 90.000,C 0.000} C_DIS
LIN {X -45.181,Y -7.308,Z -192.070,A -90.000,B 90.000,C 0.000} C_DIS
LIN {X -44.950,Y -7.308,Z -191.921,A -90.000,B 90.000,C 0.000} C_DIS
LIN {X -41.062,Y -7.308,Z -189.298,A -90.000,B 90.000,C 0.000} C_DIS
LIN {X -40.958,Y -7.308,Z -189.227,A -90.000,B 90.000,C 0.000} C_DIS
LIN {X -37.563,Y -7.308,Z -186.826,A -90.000,B 90.000,C 0.000} C_DIS
LIN {X -37.477,Y -7.308,Z -186.765,A -90.000,B 90.000,C 0.000} C_DIS
LIN {X -37.399,Y -7.308,Z -186.708,A -90.000,B 90.000,C 0.000} C_DIS
LIN {X -37.399,Y -7.308,Z -186.707,A -90.000,B 90.000,C 0.000} C_DIS
LIN {X -36.788,Y -7.308,Z -186.261,A -90.000,B 90.000,C 0.000} C_DIS
LIN {X -36.691,Y -7.308,Z -186.190,A -90.000,B 90.000,C 0.000} C_DIS
LIN {X -34.262,Y -7.308,Z -184.416,A -90.000,B 90.000,C 0.000} C_DIS
LIN {X -34.153,Y -7.308,Z -184.332,A -90.000,B 90.000,C 0.000} C_DIS
LIN {X -31.654,Y -7.308,Z -182.423,A -90.000,B 90.000,C 0.000} C_DIS
LIN {X -31.543,Y -7.308,Z -182.333,A -90.000,B 90.000,C 0.000} C_DIS
LIN {X -31.509,Y -7.308,Z -182.304,A -90.000,B 90.000,C 0.000} C_DIS
LIN {X -29.021,Y -7.308,Z -180.285,A -90.000,B 90.000,C 0.000} C_DIS
LIN {X -28.836,Y -7.308,Z -180.122,A -90.000,B 90.000,C 0.000} C_DIS
LIN {X -28.830,Y -7.308,Z -180.117,A -90.000,B 90.000,C 0.000} C_DIS
LIN {X -28.809,Y -7.308,Z -180.099,A -90.000,B 90.000,C 0.000} C_DIS
LIN {X -26.719,Y -7.308,Z -178.263,A -90.000,B 90.000,C 0.000} C_DIS
LIN {X -25.136,Y -7.308,Z -176.724,A -90.000,B 90.000,C 0.000} C_DIS
LIN {X -24.884,Y -7.308,Z -176.479,A -90.000,B 90.000,C 0.000} C_DIS
LIN {X -23.457,Y -7.308,Z -174.905,A -90.000,B 90.000,C 0.000} C_DIS
LIN {X -23.293,Y -7.308,Z -174.725,A -90.000,B 90.000,C 0.000} C_DIS
LIN {X -23.206,Y -7.308,Z -174.630,A -90.000,B 90.000,C 0.000} C_DIS
LIN {X -21.968,Y -7.308,Z -173.053,A -90.000,B 90.000,C 0.000} C_DIS
LIN {X -21.724,Y -7.308,Z -172.749,A -90.000,B 90.000,C 0.000} C_DIS
LIN {X -20.769,Y -7.308,Z -171.330,A -90.000,B 90.000,C 0.000} C_DIS
LIN {X -20.718,Y -7.308,Z -171.255,A -90.000,B 90.000,C 0.000} C_DIS
LIN {X -20.717,Y -7.308,Z -171.254,A -90.000,B 90.000,C 0.000} C_DIS
LIN {X -20.695,Y -7.308,Z -171.222,A -90.000,B 90.000,C 0.000} C_DIS
LIN {X -20.523,Y -7.308,Z -170.970,A -90.000,B 90.000,C 0.000} C_DIS
LIN {X -20.510,Y -7.308,Z -170.951,A -90.000,B 90.000,C 0.000} C_DIS
LIN {X -20.510,Y -7.308,Z -170.950,A -90.000,B 90.000,C 0.000} C_DIS
LIN {X -20.460,Y -7.308,Z -170.876,A -90.000,B 90.000,C 0.000} C_DIS
LIN {X -20.459,Y -7.308,Z -170.875,A -90.000,B 90.000,C 0.000} C_DIS
LIN {X -19.983,Y -7.308,Z -170.054,A -90.000,B 90.000,C 0.000} C_DIS
LIN {X -19.166,Y -7.308,Z -168.647,A -90.000,B 90.000,C 0.000} C_DIS
LIN {X -19.162,Y -7.308,Z -168.639,A -90.000,B 90.000,C 0.000} C_DIS
LIN {X -19.091,Y -7.308,Z -168.500,A -90.000,B 90.000,C 0.000} C_DIS
LIN {X -19.081,Y -7.308,Z -168.480,A -90.000,B 90.000,C 0.000} C_DIS
LIN {X -19.043,Y -7.308,Z -168.403,A -90.000,B 90.000,C 0.000} C_DIS
LIN {X -19.035,Y -7.308,Z -168.388,A -90.000,B 90.000,C 0.000} C_DIS
LIN {X -18.146,Y -7.308,Z -166.610,A -90.000,B 90.000,C 0.000} C_DIS
LIN {X -18.144,Y -7.308,Z -166.606,A -90.000,B 90.000,C 0.000} C_DIS
LIN {X -17.985,Y -7.308,Z -166.224,A -90.000,B 90.000,C 0.000} C_DIS
LIN {X -17.984,Y -7.308,Z -166.222,A -90.000,B 90.000,C 0.000} C_DIS
LIN {X -17.962,Y -7.308,Z -166.170,A -90.000,B 90.000,C 0.000} C_DIS
LIN {X -17.284,Y -7.308,Z -164.546,A -90.000,B 90.000,C 0.000} C_DIS
LIN {X -17.196,Y -7.308,Z -164.253,A -90.000,B 90.000,C 0.000} C_DIS
LIN {X -17.195,Y -7.308,Z -164.251,A -90.000,B 90.000,C 0.000} C_DIS
LIN {X -17.171,Y -7.308,Z -164.172,A -90.000,B 90.000,C 0.000} C_DIS
LIN {X -17.137,Y -7.308,Z -164.063,A -90.000,B 90.000,C 0.000} C_DIS
LIN {X -16.865,Y -7.308,Z -163.195,A -90.000,B 90.000,C 0.000} C_DIS
LIN {X -16.802,Y -7.308,Z -162.995,A -90.000,B 90.000,C 0.000} C_DIS
LIN {X -16.795,Y -7.308,Z -162.947,A -90.000,B 90.000,C 0.000} C_DIS
LIN {X -16.792,Y -7.308,Z -162.928,A -90.000,B 90.000,C 0.000} C_DIS
LIN {X -16.750,Y -7.308,Z -162.654,A -90.000,B 90.000,C 0.000} C_DIS
LIN {X -16.741,Y -7.308,Z -162.590,A -90.000,B 90.000,C 0.000} C_DIS
LIN {X -16.732,Y -7.308,Z -162.533,A -90.000,B 90.000,C 0.000} C_DIS
LIN {X -16.706,Y -7.308,Z -162.365,A -90.000,B 90.000,C 0.000} C_DIS
LIN {X -16.699,Y -7.308,Z -162.320,A -90.000,B 90.000,C 0.000} C_DIS
LIN {X -16.699,Y -7.308,Z -162.317,A -90.000,B 90.000,C 0.000} C_DIS
LIN {X -16.673,Y -7.308,Z -162.145,A -90.000,B 90.000,C 0.000} C_DIS
LIN {X -16.681,Y -7.308,Z -162.004,A -90.000,B 90.000,C 0.000} C_DIS
LIN {X -16.682,Y -7.308,Z -161.994,A -90.000,B 90.000,C 0.000} C_DIS
LIN {X -16.685,Y -7.308,Z -161.949,A -90.000,B 90.000,C 0.000} C_DIS
LIN {X -16.690,Y -7.308,Z -161.845,A -90.000,B 90.000,C 0.000} C_DIS
LIN {X -16.691,Y -7.308,Z -161.821,A -90.000,B 90.000,C 0.000} C_DIS
LIN {X -16.698,Y -7.308,Z -161.662,A -90.000,B 90.000,C 0.000} C_DIS
LIN {X -16.714,Y -7.308,Z -161.605,A -90.000,B 90.000,C 0.000} C_DIS
LIN {X -16.719,Y -7.308,Z -161.586,A -90.000,B 90.000,C 0.000} C_DIS
LIN {X -16.747,Y -7.308,Z -161.477,A -90.000,B 90.000,C 0.000} C_DIS
LIN {X -16.787,Y -7.308,Z -161.316,A -90.000,B 90.000,C 0.000} C_DIS
LIN {X -16.818,Y -7.308,Z -161.195,A -90.000,B 90.000,C 0.000} C_DIS
LIN {X -16.891,Y -7.308,Z -161.012,A -90.000,B 90.000,C 0.000} C_DIS
LIN {X -17.133,Y -7.308,Z -160.410,A -90.000,B 90.000,C 0.000} C_DIS
LIN {X -17.223,Y -7.308,Z -160.234,A -90.000,B 90.000,C 0.000} C_DIS
LIN {X -17.253,Y -7.308,Z -160.176,A -90.000,B 90.000,C 0.000} C_DIS
LIN {X -17.262,Y -7.308,Z -160.157,A -90.000,B 90.000,C 0.000} C_DIS
LIN {X -17.593,Y -7.308,Z -159.417,A -90.000,B 90.000,C 0.000} C_DIS
LIN {X -17.678,Y -7.308,Z -159.281,A -90.000,B 90.000,C 0.000} C_DIS
LIN {X -17.682,Y -7.308,Z -159.274,A -90.000,B 90.000,C 0.000} C_DIS
LIN {X -17.719,Y -7.308,Z -159.212,A -90.000,B 90.000,C 0.000} C_DIS
LIN {X -17.773,Y -7.308,Z -159.122,A -90.000,B 90.000,C 0.000} C_DIS
LIN {X -17.815,Y -7.308,Z -159.050,A -90.000,B 90.000,C 0.000} C_DIS
LIN {X -17.893,Y -7.308,Z -158.919,A -90.000,B 90.000,C 0.000} C_DIS
LIN {X -17.916,Y -7.308,Z -158.879,A -90.000,B 90.000,C 0.000} C_DIS
LIN {X -17.928,Y -7.308,Z -158.859,A -90.000,B 90.000,C 0.000} C_DIS
LIN {X -17.943,Y -7.308,Z -158.833,A -90.000,B 90.000,C 0.000} C_DIS
LIN {X -18.224,Y -7.308,Z -158.334,A -90.000,B 90.000,C 0.000} C_DIS
LIN {X -18.396,Y -7.308,Z -158.107,A -90.000,B 90.000,C 0.000} C_DIS
LIN {X -18.441,Y -7.308,Z -158.047,A -90.000,B 90.000,C 0.000} C_DIS
LIN {X -18.503,Y -7.308,Z -157.963,A -90.000,B 90.000,C 0.000} C_DIS
LIN {X -18.517,Y -7.308,Z -157.944,A -90.000,B 90.000,C 0.000} C_DIS
LIN {X -18.684,Y -7.308,Z -157.720,A -90.000,B 90.000,C 0.000} C_DIS
LIN {X -18.715,Y -7.308,Z -157.675,A -90.000,B 90.000,C 0.000} C_DIS
LIN {X -18.716,Y -7.308,Z -157.674,A -90.000,B 90.000,C 0.000} C_DIS
LIN {X -19.239,Y -7.308,Z -156.932,A -90.000,B 90.000,C 0.000} C_DIS
LIN {X -19.878,Y -7.308,Z -156.210,A -90.000,B 90.000,C 0.000} C_DIS
LIN {X -19.928,Y -7.308,Z -156.150,A -90.000,B 90.000,C 0.000} C_DIS
LIN {X -20.855,Y -7.308,Z -155.045,A -90.000,B 90.000,C 0.000} C_DIS
LIN {X -21.658,Y -7.308,Z -154.233,A -90.000,B 90.000,C 0.000} C_DIS
LIN {X -21.864,Y -7.308,Z -154.019,A -90.000,B 90.000,C 0.000} C_DIS
LIN {X -21.890,Y -7.308,Z -153.993,A -90.000,B 90.000,C 0.000} C_DIS
LIN {X -22.005,Y -7.308,Z -153.874,A -90.000,B 90.000,C 0.000} C_DIS
LIN {X -22.171,Y -7.308,Z -153.702,A -90.000,B 90.000,C 0.000} C_DIS
LIN {X -22.177,Y -7.308,Z -153.695,A -90.000,B 90.000,C 0.000} C_DIS
LIN {X -22.201,Y -7.308,Z -153.670,A -90.000,B 90.000,C 0.000} C_DIS
LIN {X -23.330,Y -7.308,Z -152.485,A -90.000,B 90.000,C 0.000} C_DIS
LIN {X -24.954,Y -7.308,Z -150.831,A -90.000,B 90.000,C 0.000} C_DIS
LIN {X -26.335,Y -7.308,Z -149.384,A -90.000,B 90.000,C 0.000} C_DIS
LIN {X -28.020,Y -7.308,Z -147.529,A -90.000,B 90.000,C 0.000} C_DIS
LIN {X -29.478,Y -7.308,Z -145.886,A -90.000,B 90.000,C 0.000} C_DIS
LIN {X -29.647,Y -7.308,Z -145.690,A -90.000,B 90.000,C 0.000} C_DIS
LIN {X -29.795,Y -7.308,Z -145.518,A -90.000,B 90.000,C 0.000} C_DIS
LIN {X -31.421,Y -7.308,Z -143.449,A -90.000,B 90.000,C 0.000} C_DIS
LIN {X -32.785,Y -7.308,Z -141.681,A -90.000,B 90.000,C 0.000} C_DIS
LIN {X -32.937,Y -7.308,Z -141.463,A -90.000,B 90.000,C 0.000} C_DIS
LIN {X -33.063,Y -7.308,Z -141.282,A -90.000,B 90.000,C 0.000} C_DIS
LIN {X -34.181,Y -7.308,Z -139.459,A -90.000,B 90.000,C 0.000} C_DIS
LIN {X -35.606,Y -7.308,Z -137.168,A -90.000,B 90.000,C 0.000} C_DIS
LIN {X -35.744,Y -7.308,Z -136.919,A -90.000,B 90.000,C 0.000} C_DIS
LIN {X -35.842,Y -7.308,Z -136.742,A -90.000,B 90.000,C 0.000} C_DIS
LIN {X -36.688,Y -7.308,Z -135.100,A -90.000,B 90.000,C 0.000} C_DIS
LIN {X -37.966,Y -7.308,Z -132.641,A -90.000,B 90.000,C 0.000} C_DIS
LIN {X -38.560,Y -7.308,Z -131.338,A -90.000,B 90.000,C 0.000} C_DIS
LIN {X -39.700,Y -7.308,Z -128.840,A -90.000,B 90.000,C 0.000} C_DIS
LIN {X -40.078,Y -7.308,Z -127.954,A -90.000,B 90.000,C 0.000} C_DIS
LIN {X -40.217,Y -7.308,Z -127.629,A -90.000,B 90.000,C 0.000} C_DIS
LIN {X -40.269,Y -7.308,Z -127.507,A -90.000,B 90.000,C 0.000} C_DIS
LIN {X -41.083,Y -7.308,Z -125.592,A -90.000,B 90.000,C 0.000} C_DIS
LIN {X -41.931,Y -7.308,Z -123.668,A -90.000,B 90.000,C 0.000} C_DIS
LIN {X -41.955,Y -7.308,Z -123.612,A -90.000,B 90.000,C 0.000} C_DIS
LIN {X -42.108,Y -7.308,Z -123.269,A -90.000,B 90.000,C 0.000} C_DIS
LIN {X -42.865,Y -7.308,Z -121.734,A -90.000,B 90.000,C 0.000} C_DIS
LIN {X -42.866,Y -7.308,Z -121.733,A -90.000,B 90.000,C 0.000} C_DIS
LIN {X -42.910,Y -7.308,Z -121.643,A -90.000,B 90.000,C 0.000} C_DIS
LIN {X -43.668,Y -7.308,Z -120.366,A -90.000,B 90.000,C 0.000} C_DIS
LIN {X -43.672,Y -7.308,Z -120.360,A -90.000,B 90.000,C 0.000} C_DIS
LIN {X -43.683,Y -7.308,Z -120.341,A -90.000,B 90.000,C 0.000} C_DIS
LIN {X -43.685,Y -7.308,Z -120.339,A -90.000,B 90.000,C 0.000} C_DIS
LIN {X -44.562,Y -7.308,Z -119.087,A -90.000,B 90.000,C 0.000} C_DIS
LIN {X -45.929,Y -7.308,Z -117.318,A -90.000,B 90.000,C 0.000} C_DIS
LIN {X -46.129,Y -7.308,Z -117.063,A -90.000,B 90.000,C 0.000} C_DIS
LIN {X -47.663,Y -7.308,Z -115.154,A -90.000,B 90.000,C 0.000} C_DIS
LIN {X -48.032,Y -7.308,Z -114.703,A -90.000,B 90.000,C 0.000} C_DIS
LIN {X -49.607,Y -7.308,Z -112.756,A -90.000,B 90.000,C 0.000} C_DIS
LIN {X -50.183,Y -7.308,Z -112.055,A -90.000,B 90.000,C 0.000} C_DIS
LIN {X -51.674,Y -7.308,Z -110.188,A -90.000,B 90.000,C 0.000} C_DIS
LIN {X -52.492,Y -7.308,Z -109.168,A -90.000,B 90.000,C 0.000} C_DIS
LIN {X -53.606,Y -7.308,Z -107.713,A -90.000,B 90.000,C 0.000} C_DIS
LIN {X -54.857,Y -7.308,Z -106.093,A -90.000,B 90.000,C 0.000} C_DIS
LIN {X -56.389,Y -7.308,Z -104.074,A -90.000,B 90.000,C 0.000} C_DIS
LIN {X -57.242,Y -7.308,Z -102.970,A -90.000,B 90.000,C 0.000} C_DIS
LIN {X -59.187,Y -7.308,Z -100.478,A -90.000,B 90.000,C 0.000} C_DIS
LIN {X -59.235,Y -7.308,Z -100.416,A -90.000,B 90.000,C 0.000} C_DIS
LIN {X -59.535,Y -7.308,Z -100.040,A -90.000,B 90.000,C 0.000} C_DIS
LIN {X -59.560,Y -7.308,Z -100.011,A -90.000,B 90.000,C 0.000} C_DIS
LIN {X -60.998,Y -7.308,Z -98.295,A -90.000,B 90.000,C 0.000} C_DIS
LIN {X -61.028,Y -7.308,Z -98.259,A -90.000,B 90.000,C 0.000} C_DIS
LIN {X -61.075,Y -7.308,Z -98.202,A -90.000,B 90.000,C 0.000} C_DIS
LIN {X -61.091,Y -7.308,Z -98.184,A -90.000,B 90.000,C 0.000} C_DIS
LIN {X -61.130,Y -7.308,Z -98.139,A -90.000,B 90.000,C 0.000} C_DIS
LIN {X -61.632,Y -7.308,Z -97.555,A -90.000,B 90.000,C 0.000} C_DIS
LIN {X -62.017,Y -7.308,Z -97.163,A -90.000,B 90.000,C 0.000} C_DIS
LIN {X -62.069,Y -7.308,Z -97.108,A -90.000,B 90.000,C 0.000} C_DIS
LIN {X -62.124,Y -7.308,Z -97.051,A -90.000,B 90.000,C 0.000} C_DIS
LIN {X -63.759,Y -7.308,Z -95.333,A -90.000,B 90.000,C 0.000} C_DIS
LIN {X -63.767,Y -7.308,Z -95.325,A -90.000,B 90.000,C 0.000} C_DIS
LIN {X -64.013,Y -7.308,Z -95.105,A -90.000,B 90.000,C 0.000} C_DIS
LIN {X -64.273,Y -7.308,Z -94.868,A -90.000,B 90.000,C 0.000} C_DIS
LIN {X -64.283,Y -7.308,Z -94.858,A -90.000,B 90.000,C 0.000} C_DIS
LIN {X -64.350,Y -7.308,Z -94.797,A -90.000,B 90.000,C 0.000} C_DIS
LIN {X -64.402,Y -7.308,Z -94.750,A -90.000,B 90.000,C 0.000} C_DIS
LIN {X -65.773,Y -7.308,Z -93.487,A -90.000,B 90.000,C 0.000} C_DIS
LIN {X -65.777,Y -7.308,Z -93.484,A -90.000,B 90.000,C 0.000} C_DIS
LIN {X -66.079,Y -7.308,Z -93.242,A -90.000,B 90.000,C 0.000} C_DIS
LIN {X -66.141,Y -7.308,Z -93.192,A -90.000,B 90.000,C 0.000} C_DIS
LIN {X -66.180,Y -7.308,Z -93.161,A -90.000,B 90.000,C 0.000} C_DIS
LIN {X -66.468,Y -7.308,Z -92.930,A -90.000,B 90.000,C 0.000} C_DIS
LIN {X -67.729,Y -7.308,Z -91.902,A -90.000,B 90.000,C 0.000} C_DIS
LIN {X -68.230,Y -7.308,Z -91.539,A -90.000,B 90.000,C 0.000} C_DIS
LIN {X -68.302,Y -7.308,Z -91.486,A -90.000,B 90.000,C 0.000} C_DIS
LIN {X -69.877,Y -7.308,Z -90.327,A -90.000,B 90.000,C 0.000} C_DIS
LIN {X -71.498,Y -7.308,Z -89.216,A -90.000,B 90.000,C 0.000} C_DIS
LIN {X -72.119,Y -7.308,Z -88.797,A -90.000,B 90.000,C 0.000} C_DIS
LIN {X -73.479,Y -7.308,Z -87.911,A -90.000,B 90.000,C 0.000} C_DIS
LIN {X -73.510,Y -7.308,Z -87.891,A -90.000,B 90.000,C 0.000} C_DIS
LIN {X -74.185,Y -7.308,Z -87.458,A -90.000,B 90.000,C 0.000} C_DIS
LIN {X -74.214,Y -7.308,Z -87.440,A -90.000,B 90.000,C 0.000} C_DIS
LIN {X -74.945,Y -7.308,Z -86.977,A -90.000,B 90.000,C 0.000} C_DIS
LIN {X -75.934,Y -7.308,Z -86.358,A -90.000,B 90.000,C 0.000} C_DIS
LIN {X -76.597,Y -7.308,Z -85.938,A -90.000,B 90.000,C 0.000} C_DIS
LIN {X -77.764,Y -7.308,Z -85.204,A -90.000,B 90.000,C 0.000} C_DIS
LIN {X -77.856,Y -7.308,Z -85.145,A -90.000,B 90.000,C 0.000} C_DIS
LIN {X -78.166,Y -7.308,Z -84.948,A -90.000,B 90.000,C 0.000} C_DIS
LIN {X -78.471,Y -7.308,Z -84.747,A -90.000,B 90.000,C 0.000} C_DIS
LIN {X -79.723,Y -7.308,Z -83.917,A -90.000,B 90.000,C 0.000} C_DIS
LIN {X -79.776,Y -7.308,Z -83.880,A -90.000,B 90.000,C 0.000} C_DIS
LIN {X -80.107,Y -7.308,Z -83.647,A -90.000,B 90.000,C 0.000} C_DIS
LIN {X -80.928,Y -7.308,Z -83.065,A -90.000,B 90.000,C 0.000} C_DIS
LIN {X -81.067,Y -7.308,Z -82.965,A -90.000,B 90.000,C 0.000} C_DIS
LIN {X -81.987,Y -7.308,Z -82.269,A -90.000,B 90.000,C 0.000} C_DIS
LIN {X -82.255,Y -7.308,Z -82.065,A -90.000,B 90.000,C 0.000} C_DIS
LIN {X -82.536,Y -7.308,Z -81.843,A -90.000,B 90.000,C 0.000} C_DIS
LIN {X -82.628,Y -7.308,Z -81.769,A -90.000,B 90.000,C 0.000} C_DIS
LIN {X -83.368,Y -7.308,Z -81.173,A -90.000,B 90.000,C 0.000} C_DIS
LIN {X -83.713,Y -7.308,Z -80.897,A -90.000,B 90.000,C 0.000} C_DIS
LIN {X -84.082,Y -7.308,Z -80.591,A -90.000,B 90.000,C 0.000} C_DIS
LIN {X -84.747,Y -7.308,Z -80.028,A -90.000,B 90.000,C 0.000} C_DIS
LIN {X -85.143,Y -7.308,Z -79.697,A -90.000,B 90.000,C 0.000} C_DIS
LIN {X -85.732,Y -7.308,Z -79.188,A -90.000,B 90.000,C 0.000} C_DIS
LIN {X -86.110,Y -7.308,Z -78.876,A -90.000,B 90.000,C 0.000} C_DIS
LIN {X -86.127,Y -7.308,Z -78.862,A -90.000,B 90.000,C 0.000} C_DIS
LIN {X -86.649,Y -7.308,Z -78.419,A -90.000,B 90.000,C 0.000} C_DIS
LIN {X -86.680,Y -7.308,Z -78.395,A -90.000,B 90.000,C 0.000} C_DIS
LIN {X -86.681,Y -7.308,Z -78.394,A -90.000,B 90.000,C 0.000} C_DIS
LIN {X -86.894,Y -7.308,Z -78.225,A -90.000,B 90.000,C 0.000} C_DIS
LIN {X -86.922,Y -7.308,Z -78.203,A -90.000,B 90.000,C 0.000} C_DIS
LIN {X -87.052,Y -7.308,Z -78.099,A -90.000,B 90.000,C 0.000} C_DIS
LIN {X -87.220,Y -7.308,Z -77.965,A -90.000,B 90.000,C 0.000} C_DIS
LIN {X -87.560,Y -7.308,Z -77.718,A -90.000,B 90.000,C 0.000} C_DIS
LIN {X -87.567,Y -7.308,Z -77.713,A -90.000,B 90.000,C 0.000} C_DIS
LIN {X -87.568,Y -7.308,Z -77.712,A -90.000,B 90.000,C 0.000} C_DIS
LIN {X -88.016,Y -7.308,Z -77.395,A -90.000,B 90.000,C 0.000} C_DIS
LIN {X -88.042,Y -7.308,Z -77.377,A -90.000,B 90.000,C 0.000} C_DIS
LIN {X -88.066,Y -7.308,Z -77.359,A -90.000,B 90.000,C 0.000} C_DIS
LIN {X -88.159,Y -7.308,Z -77.298,A -90.000,B 90.000,C 0.000} C_DIS
LIN {X -88.269,Y -7.308,Z -77.226,A -90.000,B 90.000,C 0.000} C_DIS
LIN {X -88.307,Y -7.308,Z -77.201,A -90.000,B 90.000,C 0.000} C_DIS
LIN {X -88.326,Y -7.308,Z -77.188,A -90.000,B 90.000,C 0.000} C_DIS
LIN {X -88.328,Y -7.308,Z -77.188,A -90.000,B 90.000,C 0.000} C_DIS
LIN {X -88.487,Y -7.308,Z -77.088,A -90.000,B 90.000,C 0.000} C_DIS
LIN {X -88.793,Y -7.308,Z -76.906,A -90.000,B 90.000,C 0.000} C_DIS
LIN {X -88.814,Y -7.308,Z -76.894,A -90.000,B 90.000,C 0.000} C_DIS
LIN {X -89.226,Y -7.308,Z -76.665,A -90.000,B 90.000,C 0.000} C_DIS
LIN {X -89.254,Y -7.308,Z -76.650,A -90.000,B 90.000,C 0.000} C_DIS
LIN {X -89.260,Y -7.308,Z -76.646,A -90.000,B 90.000,C 0.000} C_DIS
LIN {X -89.265,Y -7.308,Z -76.644,A -90.000,B 90.000,C 0.000} C_DIS
LIN {X -89.403,Y -7.308,Z -76.572,A -90.000,B 90.000,C 0.000} C_DIS
LIN {X -89.483,Y -7.308,Z -76.530,A -90.000,B 90.000,C 0.000} C_DIS
LIN {X -89.549,Y -7.308,Z -76.498,A -90.000,B 90.000,C 0.000} C_DIS
LIN {X -89.594,Y -7.308,Z -76.478,A -90.000,B 90.000,C 0.000} C_DIS
LIN {X -89.818,Y -7.308,Z -76.383,A -90.000,B 90.000,C 0.000} C_DIS
LIN {X -89.866,Y -7.308,Z -76.362,A -90.000,B 90.000,C 0.000} C_DIS
LIN {X -90.061,Y -7.308,Z -76.274,A -90.000,B 90.000,C 0.000} C_DIS
LIN {X -90.078,Y -7.308,Z -76.267,A -90.000,B 90.000,C 0.000} C_DIS
LIN {X -90.101,Y -7.308,Z -76.256,A -90.000,B 90.000,C 0.000} C_DIS
LIN {X -90.144,Y -7.308,Z -76.241,A -90.000,B 90.000,C 0.000} C_DIS
LIN {X -90.231,Y -7.308,Z -76.210,A -90.000,B 90.000,C 0.000} C_DIS
LIN {X -90.244,Y -7.308,Z -76.206,A -90.000,B 90.000,C 0.000} C_DIS
LIN {X -90.248,Y -7.308,Z -76.204,A -90.000,B 90.000,C 0.000} C_DIS
LIN {X -90.251,Y -7.308,Z -76.204,A -90.000,B 90.000,C 0.000} C_DIS
LIN {X -90.389,Y -7.308,Z -76.170,A -90.000,B 90.000,C 0.000} C_DIS
